// TwinCAT 3 PLC project Plc
// Title: Sample PackML_V2
// Company: Beckhoff Automation GmbH
// Author: Beckhoff Automation GmbH
// ProjectVersion: 3.0.3.0
// Description: Sample PackML_V2
// ProgramVersion: 3.1.0.9
// libraries:
//   CHALET_BaseComponents, * (Beckhoff CH)
//   CHALET_Nc, * (Beckhoff CH)
//   CHALET_Vision, * (Beckhoff CH)
//   CHALET_XPlanar, * (Beckhoff CH)
//   Tc2_ControllerToolbox, * (Beckhoff Automation GmbH)
//   Tc2_EtherCAT, * (Beckhoff Automation GmbH)
//   Tc2_MC2, * (Beckhoff Automation GmbH)
//   Tc2_Standard, * (Beckhoff Automation GmbH)
//   Tc2_System, * (Beckhoff Automation GmbH)
//   Tc2_Utilities, * (Beckhoff Automation GmbH)
//   Tc3_Mc3PlanarMotion, * (Beckhoff Automation GmbH)
//   Tc3_Module, * (Beckhoff Automation GmbH)
//   Tc3_PackML_V2, * (Beckhoff Automation GmbH)
//   Tc3_Vision, * (Beckhoff Automation GmbH)
//   Tc3_XPlanarUtility, * (Beckhoff Automation GmbH & Co. KG)
// project tree:
//   COMPONENTs/ Debug.TcGVL, E_ObservationState.TcDUT, GVL_Components.TcGVL, FB_Machine.TcPOU, FB_RollingAverage_Ppm.TcPOU
//   COMPONENTs/Mode/ E_PMLMode.TcDUT, E_PMLStopReason.TcDUT
//   COMPONENTs/OEE/ ST_Analytics.TcDUT
//   COMPONENTs/PackML/ ST_PMLc_Custom.TcDUT, ST_PMLs_Custom.TcDUT, ST_PML_Custom.TcDUT
//   COMPONENTs/Unit/ FB_Unit.TcPOU
//   COMPONENTs/Vision/ E_VisionState.TcDUT, FB_VsSystem.TcPOU, I_VsSystem_Check.TcIO, I_VsSystem_Plc.TcIO
//   / PlcTask.TcTTO, VisionTask.TcTTO
//   THREADs/ PRG_ProcessCellSimulation.TcPOU, PRG_Vision.TcPOU
// real-time tasks:
//   TASK Task_Plc: cycle T#1ms, priority 5, ADS port 350
//   TASK Task_XPlanar_Hardware: cycle T#250us, priority 1, ADS port 351
//   TASK Task_XPlanar_Execute: cycle T#1ms, priority 3, ADS port 352
//   TASK Task_XPlanar_Prepare: cycle T#10ms, priority 10, ADS port 353
//   TASK Task_Job: cycle default, priority 7
//   TASK Task_Vision_Acquisition: cycle T#1ms, priority 4, ADS port 354
//   TASK Task_Vision_Display: cycle T#10ms, priority 12, ADS port 355
//   TASK Task_Vision_Execute: cycle T#10ms, priority 11, ADS port 356
//   TASK Task_IO: cycle T#50000us, priority 14, ADS port 301
//   TASK PlcTask: cycle T#10ms, priority 20, ADS port 357
//   TASK AnalyticsTask: cycle T#10ms, priority 21, ADS port 358
//   TASK AnalyticsTask_C1: cycle T#10ms, priority 22, ADS port 359
// I/O:
//   DEVICE Device 4 (USB)
//     Box 2 (C9900-L100 License-Key-USB-Stick)
//   DEVICE Device 5 (EtherCAT), AmsNetId 10.16.0.17.6.1
//     Term 1 (EK1100) [EK1100 EtherCAT Coupler (2A E-Bus)]
//       Term 2 (EK1322) [EK1322 2-port EtherCAT P junction with feed-in]
//       Term 3 (EK1322) [EK1322 2-port EtherCAT P junction with feed-in]
//         Box 19 (VCS2001-0500) [VCS2001-0500 | Area scan camera, 2.5 GBit/s, Sony IMX264, color, 5.0 MP]
//           modules: Gerät
//       Term 5 (EK1322) [EK1322 2-port EtherCAT P junction with feed-in]
//         Box 6 (VIP2000-1010) [VIP2000 Flaechenbeleuchtung, OGB-IR850, breitstrahlend, 100 x 100 mm]
//           modules: Device, Channel Infrared, Channel Blue, Channel Green, Channel Orange, Calibration Data, Calibration Data, Calibration Data, Calibration Data, Calibration Data, Calibration Data, Calibration Data, Calibration Data, Calibration Data, Calibration Data, Calibration Data, Calibration Data, Calibration Data, Calibration Data, Calibration Data, Calibration Data, Calibration Data, Calibration Data, Calibration Data, Calibration Data
//         Box 7 (VIP2000-1010) [VIP2000 Flaechenbeleuchtung, OGB-IR850, breitstrahlend, 100 x 100 mm]
//           modules: Device, Channel Infrared, Channel Blue, Channel Green, Channel Orange, Calibration Data, Calibration Data, Calibration Data, Calibration Data, Calibration Data, Calibration Data, Calibration Data, Calibration Data, Calibration Data, Calibration Data, Calibration Data, Calibration Data, Calibration Data, Calibration Data, Calibration Data, Calibration Data, Calibration Data, Calibration Data, Calibration Data, Calibration Data
//       Term 8 (EL9227-5500) [EL9227-5500 Overcurrent protection 24V DC, 2Ch., max. 10A (sum), adjustable, extended functionalities]
//       Term 9 (EL9227-9664) [EL9227-9664 Overcurrent protection 24V DC, 2Ch., 6A/4A, extended functionalities]
//       Term 11 (EL9011) [EL9011 End Terminal]
//     Box 10 (EP2316-0003) [EP2316-0003 8 Ch. Dig. In, 10µs, 8Ch. Dig. Out 24V, 0,5A, Diagnostic, 10-Pole Plug Connector]
//   DEVICE Device 2 (RT-Ethernet Adapter)
//   DEVICE Device 3 (EtherCAT), AmsNetId 10.16.0.17.4.1
//     Term 4 (APS4322-7000) [APS4322-7000 Drive]
//       Term 12 (APS4322-5000) [APS4322-5000 Feedback]
//     Term 13 (APS4322-7000) [APS4322-7000 Drive]
//       Term 14 (APS4322-5000) [APS4322-5000 Feedback]
// variable links:
//   Device 3 (EtherCAT) <-> TcCOM Objects/XPlanar/Part1/Tile1
//     Term 4 (APS4322-7000)/APS Comm Inputs/CommStatusWord <-> Data Pointer/MoverCommStatusWord
//     Term 4 (APS4322-7000)/APS Comm Inputs/Data {1..4} <-> Data Pointer/MoverCommDataIn[{0..3}]  (4 links)
//     Term 4 (APS4322-7000)/APS Comm Outputs/CommControlWord <-> Data Pointer/MoverCommControlWord
//     Term 4 (APS4322-7000)/APS Comm Outputs/Data 1 <-> Data Pointer/MoverCommDataOut
//     Term 4 (APS4322-7000)/APS Diagdata/DC Link Voltage <-> Data Pointer/DcLinkVoltage
//     Term 4 (APS4322-7000)/APS Diagdata/Power supply current <-> Data Pointer/PowerSupplyCurrent
//     Term 4 (APS4322-7000)/APS Inputs/StatusWord <-> Data Pointer/PowerUnitStatusWord
//     Term 4 (APS4322-7000)/APS Outputs/ControlWord <-> Data Pointer/PowerUnitControlWord
//     Term 4 (APS4322-7000)/APS Outputs/Current D 0X0 <-> Data Pointer/DCurrentSetPoints[0]
//     Term 4 (APS4322-7000)/APS Outputs/Current D 0X1 <-> Data Pointer/DCurrentSetPoints[1]
//     Term 4 (APS4322-7000)/APS Outputs/Current D 0X2 <-> Data Pointer/DCurrentSetPoints[2]
//     Term 4 (APS4322-7000)/APS Outputs/Current D 1X0 <-> Data Pointer/DCurrentSetPoints[6]
//     Term 4 (APS4322-7000)/APS Outputs/Current D 1X1 <-> Data Pointer/DCurrentSetPoints[7]
//     Term 4 (APS4322-7000)/APS Outputs/Current D 1X2 <-> Data Pointer/DCurrentSetPoints[8]
//     Term 4 (APS4322-7000)/APS Outputs/Current D 2X0 <-> Data Pointer/DCurrentSetPoints[12]
//     Term 4 (APS4322-7000)/APS Outputs/Current D 2X1 <-> Data Pointer/DCurrentSetPoints[13]
//     Term 4 (APS4322-7000)/APS Outputs/Current D 2X2 <-> Data Pointer/DCurrentSetPoints[14]
//     Term 4 (APS4322-7000)/APS Outputs/Current D 3X0 <-> Data Pointer/DCurrentSetPoints[18]
//     Term 4 (APS4322-7000)/APS Outputs/Current D 3X1 <-> Data Pointer/DCurrentSetPoints[19]
//     Term 4 (APS4322-7000)/APS Outputs/Current D 3X2 <-> Data Pointer/DCurrentSetPoints[20]
//     Term 4 (APS4322-7000)/APS Outputs/Current D 0Y0 <-> Data Pointer/DCurrentSetPoints[3]
//     Term 4 (APS4322-7000)/APS Outputs/Current D 0Y1 <-> Data Pointer/DCurrentSetPoints[4]
//     Term 4 (APS4322-7000)/APS Outputs/Current D 0Y2 <-> Data Pointer/DCurrentSetPoints[5]
//     Term 4 (APS4322-7000)/APS Outputs/Current D 1Y0 <-> Data Pointer/DCurrentSetPoints[9]
//     Term 4 (APS4322-7000)/APS Outputs/Current D 1Y1 <-> Data Pointer/DCurrentSetPoints[10]
//     Term 4 (APS4322-7000)/APS Outputs/Current D 1Y2 <-> Data Pointer/DCurrentSetPoints[11]
//     Term 4 (APS4322-7000)/APS Outputs/Current D 2Y0 <-> Data Pointer/DCurrentSetPoints[15]
//     Term 4 (APS4322-7000)/APS Outputs/Current D 2Y1 <-> Data Pointer/DCurrentSetPoints[16]
//     Term 4 (APS4322-7000)/APS Outputs/Current D 2Y2 <-> Data Pointer/DCurrentSetPoints[17]
//     Term 4 (APS4322-7000)/APS Outputs/Current D 3Y0 <-> Data Pointer/DCurrentSetPoints[21]
//     Term 4 (APS4322-7000)/APS Outputs/Current D 3Y1 <-> Data Pointer/DCurrentSetPoints[22]
//     Term 4 (APS4322-7000)/APS Outputs/Current D 3Y2 <-> Data Pointer/DCurrentSetPoints[23]
//     Term 4 (APS4322-7000)/APS Outputs/Current Q 0X0 <-> Data Pointer/QCurrentSetPoints[0]
//     Term 4 (APS4322-7000)/APS Outputs/Current Q 0X1 <-> Data Pointer/QCurrentSetPoints[1]
//     Term 4 (APS4322-7000)/APS Outputs/Current Q 0X2 <-> Data Pointer/QCurrentSetPoints[2]
//     Term 4 (APS4322-7000)/APS Outputs/Current Q 1X0 <-> Data Pointer/QCurrentSetPoints[6]
//     Term 4 (APS4322-7000)/APS Outputs/Current Q 1X1 <-> Data Pointer/QCurrentSetPoints[7]
//     Term 4 (APS4322-7000)/APS Outputs/Current Q 1X2 <-> Data Pointer/QCurrentSetPoints[8]
//     Term 4 (APS4322-7000)/APS Outputs/Current Q 2X0 <-> Data Pointer/QCurrentSetPoints[12]
//     Term 4 (APS4322-7000)/APS Outputs/Current Q 2X1 <-> Data Pointer/QCurrentSetPoints[13]
//     Term 4 (APS4322-7000)/APS Outputs/Current Q 2X2 <-> Data Pointer/QCurrentSetPoints[14]
//     Term 4 (APS4322-7000)/APS Outputs/Current Q 3X0 <-> Data Pointer/QCurrentSetPoints[18]
//     Term 4 (APS4322-7000)/APS Outputs/Current Q 3X1 <-> Data Pointer/QCurrentSetPoints[19]
//     Term 4 (APS4322-7000)/APS Outputs/Current Q 3X2 <-> Data Pointer/QCurrentSetPoints[20]
//     Term 4 (APS4322-7000)/APS Outputs/Current Q 0Y0 <-> Data Pointer/QCurrentSetPoints[3]
//     Term 4 (APS4322-7000)/APS Outputs/Current Q 0Y1 <-> Data Pointer/QCurrentSetPoints[4]
//     Term 4 (APS4322-7000)/APS Outputs/Current Q 0Y2 <-> Data Pointer/QCurrentSetPoints[5]
//     Term 4 (APS4322-7000)/APS Outputs/Current Q 1Y0 <-> Data Pointer/QCurrentSetPoints[9]
//     Term 4 (APS4322-7000)/APS Outputs/Current Q 1Y1 <-> Data Pointer/QCurrentSetPoints[10]
//     Term 4 (APS4322-7000)/APS Outputs/Current Q 1Y2 <-> Data Pointer/QCurrentSetPoints[11]
//     Term 4 (APS4322-7000)/APS Outputs/Current Q 2Y0 <-> Data Pointer/QCurrentSetPoints[15]
//     Term 4 (APS4322-7000)/APS Outputs/Current Q 2Y1 <-> Data Pointer/QCurrentSetPoints[16]
//     Term 4 (APS4322-7000)/APS Outputs/Current Q 2Y2 <-> Data Pointer/QCurrentSetPoints[17]
//     Term 4 (APS4322-7000)/APS Outputs/Current Q 3Y0 <-> Data Pointer/QCurrentSetPoints[21]
//     Term 4 (APS4322-7000)/APS Outputs/Current Q 3Y1 <-> Data Pointer/QCurrentSetPoints[22]
//     Term 4 (APS4322-7000)/APS Outputs/Current Q 3Y2 <-> Data Pointer/QCurrentSetPoints[23]
//     Term 4 (APS4322-7000)/APS Outputs/PhiE 0X0 <-> Data Pointer/PhiSetPoints[0]
//     Term 4 (APS4322-7000)/APS Outputs/PhiE 0X1 <-> Data Pointer/PhiSetPoints[1]
//     Term 4 (APS4322-7000)/APS Outputs/PhiE 0X2 <-> Data Pointer/PhiSetPoints[2]
//     Term 4 (APS4322-7000)/APS Outputs/PhiE 1X0 <-> Data Pointer/PhiSetPoints[6]
//     Term 4 (APS4322-7000)/APS Outputs/PhiE 1X1 <-> Data Pointer/PhiSetPoints[7]
//     Term 4 (APS4322-7000)/APS Outputs/PhiE 1X2 <-> Data Pointer/PhiSetPoints[8]
//     Term 4 (APS4322-7000)/APS Outputs/PhiE 2X0 <-> Data Pointer/PhiSetPoints[12]
//     Term 4 (APS4322-7000)/APS Outputs/PhiE 2X1 <-> Data Pointer/PhiSetPoints[13]
//     Term 4 (APS4322-7000)/APS Outputs/PhiE 2X2 <-> Data Pointer/PhiSetPoints[14]
//     Term 4 (APS4322-7000)/APS Outputs/PhiE 3X0 <-> Data Pointer/PhiSetPoints[18]
//     Term 4 (APS4322-7000)/APS Outputs/PhiE 3X1 <-> Data Pointer/PhiSetPoints[19]
//     Term 4 (APS4322-7000)/APS Outputs/PhiE 3X2 <-> Data Pointer/PhiSetPoints[20]
//     Term 4 (APS4322-7000)/APS Outputs/PhiE 0Y0 <-> Data Pointer/PhiSetPoints[3]
//     Term 4 (APS4322-7000)/APS Outputs/PhiE 0Y1 <-> Data Pointer/PhiSetPoints[4]
//     Term 4 (APS4322-7000)/APS Outputs/PhiE 0Y2 <-> Data Pointer/PhiSetPoints[5]
//     Term 4 (APS4322-7000)/APS Outputs/PhiE 1Y0 <-> Data Pointer/PhiSetPoints[9]
//     Term 4 (APS4322-7000)/APS Outputs/PhiE 1Y1 <-> Data Pointer/PhiSetPoints[10]
//     Term 4 (APS4322-7000)/APS Outputs/PhiE 1Y2 <-> Data Pointer/PhiSetPoints[11]
//     Term 4 (APS4322-7000)/APS Outputs/PhiE 2Y0 <-> Data Pointer/PhiSetPoints[15]
//     Term 4 (APS4322-7000)/APS Outputs/PhiE 2Y1 <-> Data Pointer/PhiSetPoints[16]
//     Term 4 (APS4322-7000)/APS Outputs/PhiE 2Y2 <-> Data Pointer/PhiSetPoints[17]
//     Term 4 (APS4322-7000)/APS Outputs/PhiE 3Y0 <-> Data Pointer/PhiSetPoints[21]
//     Term 4 (APS4322-7000)/APS Outputs/PhiE 3Y1 <-> Data Pointer/PhiSetPoints[22]
//     Term 4 (APS4322-7000)/APS Outputs/PhiE 3Y2 <-> Data Pointer/PhiSetPoints[23]
//     Term 4 (APS4322-7000)/Term 12 (APS4322-5000)/FB Inputs/A{0..8 step 2} X-Field <-> Data Pointer/HallSensorFieldsXYZ[{0..12 step 3}]  (5 links)
//     Term 4 (APS4322-7000)/Term 12 (APS4322-5000)/FB Inputs/A{0..8 step 2} Y-Field <-> Data Pointer/HallSensorFieldsXYZ[{1..13 step 3}]  (5 links)
//     Term 4 (APS4322-7000)/Term 12 (APS4322-5000)/FB Inputs/A{0..8 step 2} Z-Field <-> Data Pointer/HallSensorFieldsXYZ[{2..14 step 3}]  (5 links)
//     Term 4 (APS4322-7000)/Term 12 (APS4322-5000)/FB Inputs/B{1..9 step 2} X-Field <-> Data Pointer/HallSensorFieldsXYZ[{15..27 step 3}]  (5 links)
//     Term 4 (APS4322-7000)/Term 12 (APS4322-5000)/FB Inputs/B{1..9 step 2} Y-Field <-> Data Pointer/HallSensorFieldsXYZ[{16..28 step 3}]  (5 links)
//     Term 4 (APS4322-7000)/Term 12 (APS4322-5000)/FB Inputs/B{1..9 step 2} Z-Field <-> Data Pointer/HallSensorFieldsXYZ[{17..29 step 3}]  (5 links)
//     Term 4 (APS4322-7000)/Term 12 (APS4322-5000)/FB Inputs/C{0..8 step 2} X-Field <-> Data Pointer/HallSensorFieldsXYZ[{30..42 step 3}]  (5 links)
//     Term 4 (APS4322-7000)/Term 12 (APS4322-5000)/FB Inputs/C{0..8 step 2} Y-Field <-> Data Pointer/HallSensorFieldsXYZ[{31..43 step 3}]  (5 links)
//     Term 4 (APS4322-7000)/Term 12 (APS4322-5000)/FB Inputs/C{0..8 step 2} Z-Field <-> Data Pointer/HallSensorFieldsXYZ[{32..44 step 3}]  (5 links)
//     Term 4 (APS4322-7000)/Term 12 (APS4322-5000)/FB Inputs/D{1..9 step 2} X-Field <-> Data Pointer/HallSensorFieldsXYZ[{45..57 step 3}]  (5 links)
//     Term 4 (APS4322-7000)/Term 12 (APS4322-5000)/FB Inputs/D{1..9 step 2} Y-Field <-> Data Pointer/HallSensorFieldsXYZ[{46..58 step 3}]  (5 links)
//     Term 4 (APS4322-7000)/Term 12 (APS4322-5000)/FB Inputs/D{1..9 step 2} Z-Field <-> Data Pointer/HallSensorFieldsXYZ[{47..59 step 3}]  (5 links)
//     Term 4 (APS4322-7000)/Term 12 (APS4322-5000)/FB Inputs/E{0..8 step 2} X-Field <-> Data Pointer/HallSensorFieldsXYZ[{60..72 step 3}]  (5 links)
//     Term 4 (APS4322-7000)/Term 12 (APS4322-5000)/FB Inputs/E{0..8 step 2} Y-Field <-> Data Pointer/HallSensorFieldsXYZ[{61..73 step 3}]  (5 links)
//     Term 4 (APS4322-7000)/Term 12 (APS4322-5000)/FB Inputs/E{0..8 step 2} Z-Field <-> Data Pointer/HallSensorFieldsXYZ[{62..74 step 3}]  (5 links)
//     Term 4 (APS4322-7000)/Term 12 (APS4322-5000)/FB Inputs/F{1..9 step 2} X-Field <-> Data Pointer/HallSensorFieldsXYZ[{75..87 step 3}]  (5 links)
//     Term 4 (APS4322-7000)/Term 12 (APS4322-5000)/FB Inputs/F{1..9 step 2} Y-Field <-> Data Pointer/HallSensorFieldsXYZ[{76..88 step 3}]  (5 links)
//     Term 4 (APS4322-7000)/Term 12 (APS4322-5000)/FB Inputs/F{1..9 step 2} Z-Field <-> Data Pointer/HallSensorFieldsXYZ[{77..89 step 3}]  (5 links)
//     Term 4 (APS4322-7000)/Term 12 (APS4322-5000)/FB Inputs/G{0..8 step 2} X-Field <-> Data Pointer/HallSensorFieldsXYZ[{90..102 step 3}]  (5 links)
//     Term 4 (APS4322-7000)/Term 12 (APS4322-5000)/FB Inputs/G{0..8 step 2} Y-Field <-> Data Pointer/HallSensorFieldsXYZ[{91..103 step 3}]  (5 links)
//     Term 4 (APS4322-7000)/Term 12 (APS4322-5000)/FB Inputs/G{0..8 step 2} Z-Field <-> Data Pointer/HallSensorFieldsXYZ[{92..104 step 3}]  (5 links)
//     Term 4 (APS4322-7000)/Term 12 (APS4322-5000)/FB Inputs/H{1..9 step 2} X-Field <-> Data Pointer/HallSensorFieldsXYZ[{105..117 step 3}]  (5 links)
//     Term 4 (APS4322-7000)/Term 12 (APS4322-5000)/FB Inputs/H{1..9 step 2} Y-Field <-> Data Pointer/HallSensorFieldsXYZ[{106..118 step 3}]  (5 links)
//     Term 4 (APS4322-7000)/Term 12 (APS4322-5000)/FB Inputs/H{1..9 step 2} Z-Field <-> Data Pointer/HallSensorFieldsXYZ[{107..119 step 3}]  (5 links)
//     Term 4 (APS4322-7000)/Term 12 (APS4322-5000)/FB Inputs/I{0..8 step 2} X-Field <-> Data Pointer/HallSensorFieldsXYZ[{120..132 step 3}]  (5 links)
//     Term 4 (APS4322-7000)/Term 12 (APS4322-5000)/FB Inputs/I{0..8 step 2} Y-Field <-> Data Pointer/HallSensorFieldsXYZ[{121..133 step 3}]  (5 links)
//     Term 4 (APS4322-7000)/Term 12 (APS4322-5000)/FB Inputs/I{0..8 step 2} Z-Field <-> Data Pointer/HallSensorFieldsXYZ[{122..134 step 3}]  (5 links)
//     Term 4 (APS4322-7000)/Term 12 (APS4322-5000)/FB Inputs/J{1..9 step 2} X-Field <-> Data Pointer/HallSensorFieldsXYZ[{135..147 step 3}]  (5 links)
//     Term 4 (APS4322-7000)/Term 12 (APS4322-5000)/FB Inputs/J{1..9 step 2} Y-Field <-> Data Pointer/HallSensorFieldsXYZ[{136..148 step 3}]  (5 links)
//     Term 4 (APS4322-7000)/Term 12 (APS4322-5000)/FB Inputs/J{1..9 step 2} Z-Field <-> Data Pointer/HallSensorFieldsXYZ[{137..149 step 3}]  (5 links)
//     Term 4 (APS4322-7000)/Term 12 (APS4322-5000)/FB Inputs/Status <-> Data Pointer/FeedbackStatus
//   Device 3 (EtherCAT) <-> TcCOM Objects/XPlanar/Part1/Tile2
//     Term 13 (APS4322-7000)/APS Comm Inputs/CommStatusWord <-> Data Pointer/MoverCommStatusWord
//     Term 13 (APS4322-7000)/APS Comm Inputs/Data {1..4} <-> Data Pointer/MoverCommDataIn[{0..3}]  (4 links)
//     Term 13 (APS4322-7000)/APS Comm Outputs/CommControlWord <-> Data Pointer/MoverCommControlWord
//     Term 13 (APS4322-7000)/APS Comm Outputs/Data 1 <-> Data Pointer/MoverCommDataOut
//     Term 13 (APS4322-7000)/APS Diagdata/DC Link Voltage <-> Data Pointer/DcLinkVoltage
//     Term 13 (APS4322-7000)/APS Diagdata/Power supply current <-> Data Pointer/PowerSupplyCurrent
//     Term 13 (APS4322-7000)/APS Inputs/StatusWord <-> Data Pointer/PowerUnitStatusWord
//     Term 13 (APS4322-7000)/APS Outputs/ControlWord <-> Data Pointer/PowerUnitControlWord
//     Term 13 (APS4322-7000)/APS Outputs/Current D 0X0 <-> Data Pointer/DCurrentSetPoints[0]
//     Term 13 (APS4322-7000)/APS Outputs/Current D 0X1 <-> Data Pointer/DCurrentSetPoints[1]
//     Term 13 (APS4322-7000)/APS Outputs/Current D 0X2 <-> Data Pointer/DCurrentSetPoints[2]
//     Term 13 (APS4322-7000)/APS Outputs/Current D 1X0 <-> Data Pointer/DCurrentSetPoints[6]
//     Term 13 (APS4322-7000)/APS Outputs/Current D 1X1 <-> Data Pointer/DCurrentSetPoints[7]
//     Term 13 (APS4322-7000)/APS Outputs/Current D 1X2 <-> Data Pointer/DCurrentSetPoints[8]
//     Term 13 (APS4322-7000)/APS Outputs/Current D 2X0 <-> Data Pointer/DCurrentSetPoints[12]
//     Term 13 (APS4322-7000)/APS Outputs/Current D 2X1 <-> Data Pointer/DCurrentSetPoints[13]
//     Term 13 (APS4322-7000)/APS Outputs/Current D 2X2 <-> Data Pointer/DCurrentSetPoints[14]
//     Term 13 (APS4322-7000)/APS Outputs/Current D 3X0 <-> Data Pointer/DCurrentSetPoints[18]
//     Term 13 (APS4322-7000)/APS Outputs/Current D 3X1 <-> Data Pointer/DCurrentSetPoints[19]
//     Term 13 (APS4322-7000)/APS Outputs/Current D 3X2 <-> Data Pointer/DCurrentSetPoints[20]
//     Term 13 (APS4322-7000)/APS Outputs/Current D 0Y0 <-> Data Pointer/DCurrentSetPoints[3]
//     Term 13 (APS4322-7000)/APS Outputs/Current D 0Y1 <-> Data Pointer/DCurrentSetPoints[4]
//     Term 13 (APS4322-7000)/APS Outputs/Current D 0Y2 <-> Data Pointer/DCurrentSetPoints[5]
//     Term 13 (APS4322-7000)/APS Outputs/Current D 1Y0 <-> Data Pointer/DCurrentSetPoints[9]
//     Term 13 (APS4322-7000)/APS Outputs/Current D 1Y1 <-> Data Pointer/DCurrentSetPoints[10]
//     Term 13 (APS4322-7000)/APS Outputs/Current D 1Y2 <-> Data Pointer/DCurrentSetPoints[11]
//     Term 13 (APS4322-7000)/APS Outputs/Current D 2Y0 <-> Data Pointer/DCurrentSetPoints[15]
//     Term 13 (APS4322-7000)/APS Outputs/Current D 2Y1 <-> Data Pointer/DCurrentSetPoints[16]
//     Term 13 (APS4322-7000)/APS Outputs/Current D 2Y2 <-> Data Pointer/DCurrentSetPoints[17]
//     Term 13 (APS4322-7000)/APS Outputs/Current D 3Y0 <-> Data Pointer/DCurrentSetPoints[21]
//     Term 13 (APS4322-7000)/APS Outputs/Current D 3Y1 <-> Data Pointer/DCurrentSetPoints[22]
//     Term 13 (APS4322-7000)/APS Outputs/Current D 3Y2 <-> Data Pointer/DCurrentSetPoints[23]
//     Term 13 (APS4322-7000)/APS Outputs/Current Q 0X0 <-> Data Pointer/QCurrentSetPoints[0]
//     Term 13 (APS4322-7000)/APS Outputs/Current Q 0X1 <-> Data Pointer/QCurrentSetPoints[1]
//     Term 13 (APS4322-7000)/APS Outputs/Current Q 0X2 <-> Data Pointer/QCurrentSetPoints[2]
//     Term 13 (APS4322-7000)/APS Outputs/Current Q 1X0 <-> Data Pointer/QCurrentSetPoints[6]
//     Term 13 (APS4322-7000)/APS Outputs/Current Q 1X1 <-> Data Pointer/QCurrentSetPoints[7]
//     Term 13 (APS4322-7000)/APS Outputs/Current Q 1X2 <-> Data Pointer/QCurrentSetPoints[8]
//     Term 13 (APS4322-7000)/APS Outputs/Current Q 2X0 <-> Data Pointer/QCurrentSetPoints[12]
//     Term 13 (APS4322-7000)/APS Outputs/Current Q 2X1 <-> Data Pointer/QCurrentSetPoints[13]
//     Term 13 (APS4322-7000)/APS Outputs/Current Q 2X2 <-> Data Pointer/QCurrentSetPoints[14]
//     Term 13 (APS4322-7000)/APS Outputs/Current Q 3X0 <-> Data Pointer/QCurrentSetPoints[18]
//     Term 13 (APS4322-7000)/APS Outputs/Current Q 3X1 <-> Data Pointer/QCurrentSetPoints[19]
//     Term 13 (APS4322-7000)/APS Outputs/Current Q 3X2 <-> Data Pointer/QCurrentSetPoints[20]
//     Term 13 (APS4322-7000)/APS Outputs/Current Q 0Y0 <-> Data Pointer/QCurrentSetPoints[3]
//     Term 13 (APS4322-7000)/APS Outputs/Current Q 0Y1 <-> Data Pointer/QCurrentSetPoints[4]
//     Term 13 (APS4322-7000)/APS Outputs/Current Q 0Y2 <-> Data Pointer/QCurrentSetPoints[5]
//     Term 13 (APS4322-7000)/APS Outputs/Current Q 1Y0 <-> Data Pointer/QCurrentSetPoints[9]
//     Term 13 (APS4322-7000)/APS Outputs/Current Q 1Y1 <-> Data Pointer/QCurrentSetPoints[10]
//     Term 13 (APS4322-7000)/APS Outputs/Current Q 1Y2 <-> Data Pointer/QCurrentSetPoints[11]
//     Term 13 (APS4322-7000)/APS Outputs/Current Q 2Y0 <-> Data Pointer/QCurrentSetPoints[15]
//     Term 13 (APS4322-7000)/APS Outputs/Current Q 2Y1 <-> Data Pointer/QCurrentSetPoints[16]
//     Term 13 (APS4322-7000)/APS Outputs/Current Q 2Y2 <-> Data Pointer/QCurrentSetPoints[17]
//     Term 13 (APS4322-7000)/APS Outputs/Current Q 3Y0 <-> Data Pointer/QCurrentSetPoints[21]
//     Term 13 (APS4322-7000)/APS Outputs/Current Q 3Y1 <-> Data Pointer/QCurrentSetPoints[22]
//     Term 13 (APS4322-7000)/APS Outputs/Current Q 3Y2 <-> Data Pointer/QCurrentSetPoints[23]
//     Term 13 (APS4322-7000)/APS Outputs/PhiE 0X0 <-> Data Pointer/PhiSetPoints[0]
//     Term 13 (APS4322-7000)/APS Outputs/PhiE 0X1 <-> Data Pointer/PhiSetPoints[1]
//     Term 13 (APS4322-7000)/APS Outputs/PhiE 0X2 <-> Data Pointer/PhiSetPoints[2]
//     Term 13 (APS4322-7000)/APS Outputs/PhiE 1X0 <-> Data Pointer/PhiSetPoints[6]
//     Term 13 (APS4322-7000)/APS Outputs/PhiE 1X1 <-> Data Pointer/PhiSetPoints[7]
//     Term 13 (APS4322-7000)/APS Outputs/PhiE 1X2 <-> Data Pointer/PhiSetPoints[8]
//     Term 13 (APS4322-7000)/APS Outputs/PhiE 2X0 <-> Data Pointer/PhiSetPoints[12]
//     Term 13 (APS4322-7000)/APS Outputs/PhiE 2X1 <-> Data Pointer/PhiSetPoints[13]
//     Term 13 (APS4322-7000)/APS Outputs/PhiE 2X2 <-> Data Pointer/PhiSetPoints[14]
//     Term 13 (APS4322-7000)/APS Outputs/PhiE 3X0 <-> Data Pointer/PhiSetPoints[18]
//     Term 13 (APS4322-7000)/APS Outputs/PhiE 3X1 <-> Data Pointer/PhiSetPoints[19]
//     Term 13 (APS4322-7000)/APS Outputs/PhiE 3X2 <-> Data Pointer/PhiSetPoints[20]
//     Term 13 (APS4322-7000)/APS Outputs/PhiE 0Y0 <-> Data Pointer/PhiSetPoints[3]
//     Term 13 (APS4322-7000)/APS Outputs/PhiE 0Y1 <-> Data Pointer/PhiSetPoints[4]
//     Term 13 (APS4322-7000)/APS Outputs/PhiE 0Y2 <-> Data Pointer/PhiSetPoints[5]
//     Term 13 (APS4322-7000)/APS Outputs/PhiE 1Y0 <-> Data Pointer/PhiSetPoints[9]
//     Term 13 (APS4322-7000)/APS Outputs/PhiE 1Y1 <-> Data Pointer/PhiSetPoints[10]
//     Term 13 (APS4322-7000)/APS Outputs/PhiE 1Y2 <-> Data Pointer/PhiSetPoints[11]
//     Term 13 (APS4322-7000)/APS Outputs/PhiE 2Y0 <-> Data Pointer/PhiSetPoints[15]
//     Term 13 (APS4322-7000)/APS Outputs/PhiE 2Y1 <-> Data Pointer/PhiSetPoints[16]
//     Term 13 (APS4322-7000)/APS Outputs/PhiE 2Y2 <-> Data Pointer/PhiSetPoints[17]
//     Term 13 (APS4322-7000)/APS Outputs/PhiE 3Y0 <-> Data Pointer/PhiSetPoints[21]
//     Term 13 (APS4322-7000)/APS Outputs/PhiE 3Y1 <-> Data Pointer/PhiSetPoints[22]
//     Term 13 (APS4322-7000)/APS Outputs/PhiE 3Y2 <-> Data Pointer/PhiSetPoints[23]
//     Term 13 (APS4322-7000)/Term 14 (APS4322-5000)/FB Inputs/A{0..8 step 2} X-Field <-> Data Pointer/HallSensorFieldsXYZ[{0..12 step 3}]  (5 links)
//     Term 13 (APS4322-7000)/Term 14 (APS4322-5000)/FB Inputs/A{0..8 step 2} Y-Field <-> Data Pointer/HallSensorFieldsXYZ[{1..13 step 3}]  (5 links)
//     Term 13 (APS4322-7000)/Term 14 (APS4322-5000)/FB Inputs/A{0..8 step 2} Z-Field <-> Data Pointer/HallSensorFieldsXYZ[{2..14 step 3}]  (5 links)
//     Term 13 (APS4322-7000)/Term 14 (APS4322-5000)/FB Inputs/B{1..9 step 2} X-Field <-> Data Pointer/HallSensorFieldsXYZ[{15..27 step 3}]  (5 links)
//     Term 13 (APS4322-7000)/Term 14 (APS4322-5000)/FB Inputs/B{1..9 step 2} Y-Field <-> Data Pointer/HallSensorFieldsXYZ[{16..28 step 3}]  (5 links)
//     Term 13 (APS4322-7000)/Term 14 (APS4322-5000)/FB Inputs/B{1..9 step 2} Z-Field <-> Data Pointer/HallSensorFieldsXYZ[{17..29 step 3}]  (5 links)
//     Term 13 (APS4322-7000)/Term 14 (APS4322-5000)/FB Inputs/C{0..8 step 2} X-Field <-> Data Pointer/HallSensorFieldsXYZ[{30..42 step 3}]  (5 links)
//     Term 13 (APS4322-7000)/Term 14 (APS4322-5000)/FB Inputs/C{0..8 step 2} Y-Field <-> Data Pointer/HallSensorFieldsXYZ[{31..43 step 3}]  (5 links)
//     Term 13 (APS4322-7000)/Term 14 (APS4322-5000)/FB Inputs/C{0..8 step 2} Z-Field <-> Data Pointer/HallSensorFieldsXYZ[{32..44 step 3}]  (5 links)
//     Term 13 (APS4322-7000)/Term 14 (APS4322-5000)/FB Inputs/D{1..9 step 2} X-Field <-> Data Pointer/HallSensorFieldsXYZ[{45..57 step 3}]  (5 links)
//     Term 13 (APS4322-7000)/Term 14 (APS4322-5000)/FB Inputs/D{1..9 step 2} Y-Field <-> Data Pointer/HallSensorFieldsXYZ[{46..58 step 3}]  (5 links)
//     Term 13 (APS4322-7000)/Term 14 (APS4322-5000)/FB Inputs/D{1..9 step 2} Z-Field <-> Data Pointer/HallSensorFieldsXYZ[{47..59 step 3}]  (5 links)
//     Term 13 (APS4322-7000)/Term 14 (APS4322-5000)/FB Inputs/E{0..8 step 2} X-Field <-> Data Pointer/HallSensorFieldsXYZ[{60..72 step 3}]  (5 links)
//     Term 13 (APS4322-7000)/Term 14 (APS4322-5000)/FB Inputs/E{0..8 step 2} Y-Field <-> Data Pointer/HallSensorFieldsXYZ[{61..73 step 3}]  (5 links)
//     Term 13 (APS4322-7000)/Term 14 (APS4322-5000)/FB Inputs/E{0..8 step 2} Z-Field <-> Data Pointer/HallSensorFieldsXYZ[{62..74 step 3}]  (5 links)
//     Term 13 (APS4322-7000)/Term 14 (APS4322-5000)/FB Inputs/F{1..9 step 2} X-Field <-> Data Pointer/HallSensorFieldsXYZ[{75..87 step 3}]  (5 links)
//     Term 13 (APS4322-7000)/Term 14 (APS4322-5000)/FB Inputs/F{1..9 step 2} Y-Field <-> Data Pointer/HallSensorFieldsXYZ[{76..88 step 3}]  (5 links)
//     Term 13 (APS4322-7000)/Term 14 (APS4322-5000)/FB Inputs/F{1..9 step 2} Z-Field <-> Data Pointer/HallSensorFieldsXYZ[{77..89 step 3}]  (5 links)
//     Term 13 (APS4322-7000)/Term 14 (APS4322-5000)/FB Inputs/G{0..8 step 2} X-Field <-> Data Pointer/HallSensorFieldsXYZ[{90..102 step 3}]  (5 links)
//     Term 13 (APS4322-7000)/Term 14 (APS4322-5000)/FB Inputs/G{0..8 step 2} Y-Field <-> Data Pointer/HallSensorFieldsXYZ[{91..103 step 3}]  (5 links)
//     Term 13 (APS4322-7000)/Term 14 (APS4322-5000)/FB Inputs/G{0..8 step 2} Z-Field <-> Data Pointer/HallSensorFieldsXYZ[{92..104 step 3}]  (5 links)
//     Term 13 (APS4322-7000)/Term 14 (APS4322-5000)/FB Inputs/H{1..9 step 2} X-Field <-> Data Pointer/HallSensorFieldsXYZ[{105..117 step 3}]  (5 links)
//     Term 13 (APS4322-7000)/Term 14 (APS4322-5000)/FB Inputs/H{1..9 step 2} Y-Field <-> Data Pointer/HallSensorFieldsXYZ[{106..118 step 3}]  (5 links)
//     Term 13 (APS4322-7000)/Term 14 (APS4322-5000)/FB Inputs/H{1..9 step 2} Z-Field <-> Data Pointer/HallSensorFieldsXYZ[{107..119 step 3}]  (5 links)
//     Term 13 (APS4322-7000)/Term 14 (APS4322-5000)/FB Inputs/I{0..8 step 2} X-Field <-> Data Pointer/HallSensorFieldsXYZ[{120..132 step 3}]  (5 links)
//     Term 13 (APS4322-7000)/Term 14 (APS4322-5000)/FB Inputs/I{0..8 step 2} Y-Field <-> Data Pointer/HallSensorFieldsXYZ[{121..133 step 3}]  (5 links)
//     Term 13 (APS4322-7000)/Term 14 (APS4322-5000)/FB Inputs/I{0..8 step 2} Z-Field <-> Data Pointer/HallSensorFieldsXYZ[{122..134 step 3}]  (5 links)
//     Term 13 (APS4322-7000)/Term 14 (APS4322-5000)/FB Inputs/J{1..9 step 2} X-Field <-> Data Pointer/HallSensorFieldsXYZ[{135..147 step 3}]  (5 links)
//     Term 13 (APS4322-7000)/Term 14 (APS4322-5000)/FB Inputs/J{1..9 step 2} Y-Field <-> Data Pointer/HallSensorFieldsXYZ[{136..148 step 3}]  (5 links)
//     Term 13 (APS4322-7000)/Term 14 (APS4322-5000)/FB Inputs/J{1..9 step 2} Z-Field <-> Data Pointer/HallSensorFieldsXYZ[{137..149 step 3}]  (5 links)
//     Term 13 (APS4322-7000)/Term 14 (APS4322-5000)/FB Inputs/Status <-> Data Pointer/FeedbackStatus
//   XPlanar MC Project/Axes/Mover4220_1 <-> TcCOM Objects/XPlanar/Mover4220_1
//     IoToMc/STD <-> OutputsToNC3/HWToNC3
//   Plc/Plc Instance <-> Device 5 (EtherCAT)/Term 1 (EK1100)/Term 3 (EK1322)/Box 19 (VCS2001-0500)
//     PlcTask Outputs/GVL_Components.fbMachine.fbVsSystem.fbCameraTriggerController.nStartTime <-> Gerät/DC Timestamp/GVL_Components.fbMachine.fbVsSystem.fbCameraTriggerController.nStartTime
//   Plc/Plc Instance <-> Device 5 (EtherCAT)/Term 1 (EK1100)/Term 5 (EK1322)/Box 6 (VIP2000-1010)
//     PlcTask Inputs/GVL_Components.fbMachine.fbVsSystem.fbIllumination1.DeviceInputs/bDiag <-> VIMN Inputs Device/bDiag
//     PlcTask Inputs/GVL_Components.fbMachine.fbVsSystem.fbIllumination1.DeviceInputs/bError <-> VIMN Inputs Device/bError
//     PlcTask Inputs/GVL_Components.fbMachine.fbVsSystem.fbIllumination1.DeviceInputs/bReady <-> VIMN Inputs Device/bReady
//     PlcTask Inputs/GVL_Components.fbMachine.fbVsSystem.fbIllumination1.DeviceInputs/bWarning <-> VIMN Inputs Device/bWarning
//     PlcTask Inputs/GVL_Components.fbMachine.fbVsSystem.fbIllumination1.DeviceInputs/nSwitch_on_counter <-> VIMN Inputs Device/nSwitch_on_counter
//     PlcTask Outputs/GVL_Components.fbMachine.fbVsSystem.fbIllumination1.ChannelBlue/nBrightness <-> Channel Blue/VICH_PULSE Outputs/nBrightness
//     PlcTask Outputs/GVL_Components.fbMachine.fbVsSystem.fbIllumination1.ChannelBlue/nDuration_1us <-> Channel Blue/VICH_PULSE Outputs/nDuration_1us
//     PlcTask Outputs/GVL_Components.fbMachine.fbVsSystem.fbIllumination1.ChannelGreen/nBrightness <-> Channel Green/VICH_PULSE Outputs/nBrightness
//     PlcTask Outputs/GVL_Components.fbMachine.fbVsSystem.fbIllumination1.ChannelGreen/nDuration_1us <-> Channel Green/VICH_PULSE Outputs/nDuration_1us
//     PlcTask Outputs/GVL_Components.fbMachine.fbVsSystem.fbIllumination1.ChannelInfrared/nBrightness <-> Channel Infrared/VICH_PULSE Outputs/nBrightness
//     PlcTask Outputs/GVL_Components.fbMachine.fbVsSystem.fbIllumination1.ChannelInfrared/nDuration_1us <-> Channel Infrared/VICH_PULSE Outputs/nDuration_1us
//     PlcTask Outputs/GVL_Components.fbMachine.fbVsSystem.fbIllumination1.ChannelOrange/nBrightness <-> Channel Orange/VICH_PULSE Outputs/nBrightness
//     PlcTask Outputs/GVL_Components.fbMachine.fbVsSystem.fbIllumination1.ChannelOrange/nDuration_1us <-> Channel Orange/VICH_PULSE Outputs/nDuration_1us
//     PlcTask Outputs/GVL_Components.fbMachine.fbVsSystem.fbIllumination1.DeviceOutputs/bEnable <-> VIMN Outputs Device/bEnable
//     PlcTask Outputs/GVL_Components.fbMachine.fbVsSystem.fbIllumination1.DeviceOutputs/bReset <-> VIMN Outputs Device/bReset
//     PlcTask Outputs/GVL_Components.fbMachine.fbVsSystem.fbIllumination1.Pulse_DC_Outputs/nTimestamp <-> Device/VIOM_PULSE_DC Outputs/nTimestamp
//   Plc/Plc Instance <-> Device 5 (EtherCAT)/Term 1 (EK1100)/Term 5 (EK1322)/Box 7 (VIP2000-1010)
//     PlcTask Inputs/GVL_Components.fbMachine.fbVsSystem.fbIllumination2.DeviceInputs/bDiag <-> VIMN Inputs Device/bDiag
//     PlcTask Inputs/GVL_Components.fbMachine.fbVsSystem.fbIllumination2.DeviceInputs/bError <-> VIMN Inputs Device/bError
//     PlcTask Inputs/GVL_Components.fbMachine.fbVsSystem.fbIllumination2.DeviceInputs/bReady <-> VIMN Inputs Device/bReady
//     PlcTask Inputs/GVL_Components.fbMachine.fbVsSystem.fbIllumination2.DeviceInputs/bWarning <-> VIMN Inputs Device/bWarning
//     PlcTask Inputs/GVL_Components.fbMachine.fbVsSystem.fbIllumination2.DeviceInputs/nSwitch_on_counter <-> VIMN Inputs Device/nSwitch_on_counter
//     PlcTask Outputs/GVL_Components.fbMachine.fbVsSystem.fbIllumination2.ChannelBlue/nBrightness <-> Channel Blue/VICH_PULSE Outputs/nBrightness
//     PlcTask Outputs/GVL_Components.fbMachine.fbVsSystem.fbIllumination2.ChannelBlue/nDuration_1us <-> Channel Blue/VICH_PULSE Outputs/nDuration_1us
//     PlcTask Outputs/GVL_Components.fbMachine.fbVsSystem.fbIllumination2.ChannelGreen/nBrightness <-> Channel Green/VICH_PULSE Outputs/nBrightness
//     PlcTask Outputs/GVL_Components.fbMachine.fbVsSystem.fbIllumination2.ChannelGreen/nDuration_1us <-> Channel Green/VICH_PULSE Outputs/nDuration_1us
//     PlcTask Outputs/GVL_Components.fbMachine.fbVsSystem.fbIllumination2.ChannelInfrared/nBrightness <-> Channel Infrared/VICH_PULSE Outputs/nBrightness
//     PlcTask Outputs/GVL_Components.fbMachine.fbVsSystem.fbIllumination2.ChannelInfrared/nDuration_1us <-> Channel Infrared/VICH_PULSE Outputs/nDuration_1us
//     PlcTask Outputs/GVL_Components.fbMachine.fbVsSystem.fbIllumination2.ChannelOrange/nBrightness <-> Channel Orange/VICH_PULSE Outputs/nBrightness
//     PlcTask Outputs/GVL_Components.fbMachine.fbVsSystem.fbIllumination2.ChannelOrange/nDuration_1us <-> Channel Orange/VICH_PULSE Outputs/nDuration_1us
//     PlcTask Outputs/GVL_Components.fbMachine.fbVsSystem.fbIllumination2.DeviceOutputs/bEnable <-> VIMN Outputs Device/bEnable
//     PlcTask Outputs/GVL_Components.fbMachine.fbVsSystem.fbIllumination2.DeviceOutputs/bReset <-> VIMN Outputs Device/bReset
//     PlcTask Outputs/GVL_Components.fbMachine.fbVsSystem.fbIllumination2.Pulse_DC_Outputs/nTimestamp <-> Device/VIOM_PULSE_DC Outputs/nTimestamp
//   Plc/Plc Instance <-> XPlanar MC Project/Axes/Mover4220_1
//     PlcTask Inputs/GVL_Components.fbMachine.aMovers[1].fbMover.MCTOPLC/ACT <-> McToPlc/ACT
//     PlcTask Inputs/GVL_Components.fbMachine.aMovers[1].fbMover.MCTOPLC/COORDMODE <-> McToPlc/COORDMODE
//     PlcTask Inputs/GVL_Components.fbMachine.aMovers[1].fbMover.MCTOPLC/SET <-> McToPlc/SET
//     PlcTask Inputs/GVL_Components.fbMachine.aMovers[1].fbMover.MCTOPLC/SETONTRACK <-> McToPlc/SETONTRACK
//     PlcTask Inputs/GVL_Components.fbMachine.aMovers[1].fbMover.MCTOPLC/STD <-> McToPlc/STD
//     PlcTask Outputs/GVL_Components.fbMachine.aMovers[1].fbMover.PLCTOMC/STD <-> PlcToMc/STD
//   Plc/Plc Instance <-> XPlanar MC Project/Axes/Mover4220_2
//     PlcTask Inputs/GVL_Components.fbMachine.aMovers[2].fbMover.MCTOPLC/ACT <-> McToPlc/ACT
//     PlcTask Inputs/GVL_Components.fbMachine.aMovers[2].fbMover.MCTOPLC/COORDMODE <-> McToPlc/COORDMODE
//     PlcTask Inputs/GVL_Components.fbMachine.aMovers[2].fbMover.MCTOPLC/SET <-> McToPlc/SET
//     PlcTask Inputs/GVL_Components.fbMachine.aMovers[2].fbMover.MCTOPLC/SETONTRACK <-> McToPlc/SETONTRACK
//     PlcTask Inputs/GVL_Components.fbMachine.aMovers[2].fbMover.MCTOPLC/STD <-> McToPlc/STD
//     PlcTask Outputs/GVL_Components.fbMachine.aMovers[2].fbMover.PLCTOMC/STD <-> PlcToMc/STD
//   Plc/Plc Instance <-> XPlanar MC Project/Groups/Environment
//     PlcTask Inputs/GVL_Components.fbMachine.fbXpEnvironment.fbEnvironment.MCTOPLC_STD <-> McToPlc/STD
//   Plc/Plc Instance <-> XPlanar MC Project/Groups/Station1
//     PlcTask Inputs/GVL_Components.fbMachine.fbStation1.fbOptionalTrackUsedInLiveView.MCTOPLC_STD <-> McToPlc/STD
//   Plc/Plc Instance <-> XPlanar MC Project/Groups/Station2
//     PlcTask Inputs/GVL_Components.fbMachine.fbStation2.fbOptionalTrackUsedInLiveView.MCTOPLC_STD <-> McToPlc/STD
//   Plc/Plc Instance <-> XPlanar MC Project/Groups/Station3
//     PlcTask Inputs/GVL_Components.fbMachine.fbStation3.fbOptionalTrackUsedInLiveView.MCTOPLC_STD <-> McToPlc/STD
//   Plc/Plc Instance <-> XPlanar MC Project/Groups/Track1
//     PlcTask Inputs/GVL_Components.fbMachine.fbTrackA.fbTrack.MCTOPLC_STD <-> McToPlc/STD
//   Plc/Plc Instance <-> XPlanar MC Project/Groups/XPlanar
//     PlcTask Inputs/GVL_Components.fbMachine.fbXpGroup.fbGroup.MCTOPLC_STD <-> McToPlc/STD
//   TcCOM Objects/XPlanar/Mover4220_1 <-> XPlanar MC Project/Axes/Mover4220_1
//     InputsFromNC3/NC3ToHW <-> McToIo/STD
//   TcCOM Objects/XPlanar/Mover4220_2 <-> XPlanar MC Project/Axes/Mover4220_2
//     InputsFromNC3/NC3ToHW <-> McToIo/STD
//     OutputsToNC3/HWToNC3 <-> IoToMc/STD
//   Task_IO <-> Device 4 (USB)/Box 2 (C9900-L100 License-Key-USB-Stick)
//     Inputs/Var 2528 <-> BoxInfo/BoxState

CONFIGURATION Plc
    RESOURCE PLC ON TwinCAT3
        TASK PlcTask(INTERVAL := T#1ms, PRIORITY := 5);
        TASK VisionTask(INTERVAL := T#10ms, PRIORITY := 11);
        PROGRAM PRG_ProcessCellSimulation WITH PlcTask : PRG_ProcessCellSimulation;
        PROGRAM PRG_Vision WITH VisionTask : PRG_Vision;
    END_RESOURCE
END_CONFIGURATION

// ---- COMPONENTs/E_ObservationState.TcDUT
{attribute 'qualified_only'}
{attribute 'strict'}
TYPE E_ObservationState :
(
	Idle := 0,
	Observing,
	Qualifying,
	Done
);
END_TYPE

// ---- COMPONENTs/Mode/E_PMLMode.TcDUT
{attribute 'qualified_only'}
TYPE E_PMLMode:
(
	(* Mandatory modes *)
	UNDEFINED := 0,
	PRODUCTION := 1,
	
	(* Optional modes *)
	// MAINTANANCE := 2,
	MANUAL := 3
	
	(* Custom modes *)
	// ?? := 4..32
	// use PML_UnitModeConfig
	
) DINT := UNDEFINED;
END_TYPE

// ---- COMPONENTs/Mode/E_PMLStopReason.TcDUT
{attribute 'qualified_only'}
TYPE E_PMLStopReason :
(
	None := 0,
	Abort_EStop := 1,
	Abort_User := 2,
	Held_Material := 3,
	Held_Ingredients := 4,
	Stop_Actuators := 5,
	Stop_Sensors := 6,
	Suspend_Starved := 7,
	Suspend_Blocked := 8
) DINT := None;
END_TYPE

// ---- COMPONENTs/OEE/ST_Analytics.TcDUT
TYPE ST_Analytics :
STRUCT
	nUnitsProduced : ULINT;
	nDefectiveUnits : ULINT;
	nState : UINT;
	tMlCalculation : TIME;
	bDefectivePart : BOOL;
END_STRUCT
END_TYPE

// ---- COMPONENTs/PackML/ST_PMLc_Custom.TcDUT
TYPE ST_PMLc_Custom EXTENDS ST_PMLcMin :
STRUCT
	Parameter : ARRAY[1..2] OF ST_Descriptor;
END_STRUCT
END_TYPE

// ---- COMPONENTs/PackML/ST_PMLs_Custom.TcDUT
TYPE ST_PMLs_Custom EXTENDS ST_PMLsMin :
STRUCT
	Parameter : ARRAY [1..1] OF ST_Descriptor;
END_STRUCT
END_TYPE

// ---- COMPONENTs/PackML/ST_PML_Custom.TcDUT
TYPE ST_PML_Custom :
STRUCT
	Command 	: ST_PMLc_Custom;
	Status 		: ST_PMLs_Custom;
	Admin 		: ST_PMLaMin;
END_STRUCT
END_TYPE

// ---- COMPONENTs/Vision/E_VisionState.TcDUT
{attribute 'qualified_only'}
{attribute 'strict'}
TYPE E_VisionState :
(
	Idle := 0,
	SelectMode,
	Configure,
	Acquisition,
	Error
);
END_TYPE

// ---- COMPONENTs/Debug.TcGVL
{attribute 'qualified_only'}
VAR_GLOBAL
	tDebug : T_DCTIME64;
	tDebug2 : T_DCTIME64;
	tNow : T_DCTIME64;
END_VAR

// ---- COMPONENTs/GVL_Components.TcGVL
VAR_GLOBAL
	{attribute 'TcContextId':='0'}
	fbMachine : FB_Machine; // Process cell
END_VAR

// ---- COMPONENTs/Vision/I_VsSystem_Check.TcIO
INTERFACE I_VsSystem_Check

METHOD GetQualityRating : I_CH_Feedback
VAR_INPUT
	nDcTrigger : T_DCTIME64;
	nNbrHoles_Expected : LREAL;
	fHoleDiameter : LREAL;
END_VAR
VAR_OUTPUT
	bQualityGood : BOOL;
	nNbrHoles_Found : LREAL;
END_VAR
END_METHOD

END_INTERFACE

// ---- COMPONENTs/Vision/I_VsSystem_Plc.TcIO
INTERFACE I_VsSystem_Plc

METHOD Initialize : HRESULT
VAR_INPUT
END_VAR
END_METHOD

PROPERTY Initialized : BOOL
GET
END_GET
END_PROPERTY

METHOD Update : HRESULT
VAR_INPUT
END_VAR
END_METHOD

METHOD UpdateSlow : HRESULT
VAR_INPUT
END_VAR
END_METHOD

END_INTERFACE

// ---- THREADs/PRG_ProcessCellSimulation.TcPOU
PROGRAM PRG_ProcessCellSimulation

fbMachine.Update();

END_PROGRAM

// ---- THREADs/PRG_Vision.TcPOU
PROGRAM PRG_Vision

fbMachine.UpdateSlow();

END_PROGRAM

// ---- COMPONENTs/FB_Machine.TcPOU
{attribute 'no_explicit_call' := 'do not call this POU directly'} 
FUNCTION_BLOCK FB_Machine EXTENDS FB_Unit
VAR CONSTANT
	N_NBR_MOVERS : UINT := 2;	

	(*	Unique station identification 
		Station ID *)
	S_STATION_NAME_1 : STRING(20) := 'Load';
	S_STATION_NAME_2 : STRING(20) := 'Camera';
	S_STATION_NAME_3 : STRING(20) := 'Unload';
END_VAR
VAR
	(* 	XPlanar System - 1 per associated XPlanar 
		The system is the container and organizer for all subsequent XPlanar objects. 
		All objects are registered with this system	*)
	fbXpSystem 		: FB_XP_System();
	iXpSystem_Plc 	: I_XP_System_PLC := fbXpSystem; 
	
	(* 	XPlanar Collision Avoidance Groupe - 1 per associated XPlanar 
		The Planar group is a software object that prevents collisions between Planar movers as well as collisions of Planar movers with the boundary of 
		the stator area on the two-dimensional XPlanar stator area. To do this, the 2D areas of all objects in the group are blocked. When a motion command 
		is transferred to a mover, the required area is requested from the Planar group and the motion command is rejected if this area would collide 
		with already reserved areas. If the motion command can be executed, the area is added to the set of reserved area and blocked accordingly.	*)
	fbXpGroup : FB_XP_Group(ipSystem := fbXpSystem);
		
	(* 	XPlanar Environment - 1 per associated XPlanar 
		The Planar environment is a software object that represents the two-dimensional XPlanar stator surface. Together with Planar movers in a group, 
		it prevents collisions of the movers with the edge of the surface. *)
	fbXpEnvironment : FB_XP_Environment(ipSystem := fbXpSystem);	
	
	(* 	XPlanar mover - n per associated XPlanar. Can be instantiated as an array and/or individually
		The Planar mover is a software object that represents an XPlanar mover. It summarizes the state of the real mover (position, velocity, etc.) 
		for the user. In addition, the user has the possibility to influence or control the state of the real mover via the Planar mover. *)								
	aMovers : ARRAY[1..N_NBR_MOVERS] OF FB_XP_Mover[
		(ipSystem := fbXpSystem),
		(ipSystem := fbXpSystem)];
	
	(* 	XPlanar track - n per associated XPlanar. Can be instantiated as an array and/or individually
		The Planar track is a software object that represents a (virtual) one-dimensional path on the two-dimensional XPlanar stator surface. 
		Several Planar movers can be lined up and moved on this path. Collisions are prevented by keeping a preset distance between the movers. *)		
	fbTrackA : FB_XP_Track(ipSystem	:= fbXpSystem);	
		
	(* 	XPlanar station - n per associated XPlanar. Can be instantiated as an array and/or individually
		The stations are the main component of the application. As soon as the system has been started up and all movers are on the track, the movers are only sent from one station to the next.
		Parameters:
			xPos, yPos 			= Absolute position of the station on the xPlanar.
			ipAccocietedTrack 	= The track on which the station is located. If the XY position is not on this track, the next possible track position is assumed on this track.
			sStationID 			= Unique name that may only exist once.
			sStationGroupID 	= A name for a group to which this station belongs. Important for redundant stations
			StationAheadx 		= Which station can be approached directly from this station in the positive direction? After a switch there are several possibilities. *)		
	fbStation1	: FB_XP_Station(
					ipSystem := fbXpSystem,
					ipAccocietedTrack := fbTrackA,
					sUniqueName := S_STATION_NAME_1,
					sTargetGroup := '',
					nMoverQueueSize	:= 1,
					xPos := 120,
					yPos := 60);
							
	fbStation2 	: FB_XP_Station(
					ipSystem := fbXpSystem,
					ipAccocietedTrack := fbTrackA,
					sUniqueName := S_STATION_NAME_2,
					sTargetGroup := '',
					nMoverQueueSize := 1,
					xPos := 60,
					yPos := 240);			
	
	fbStation3 	: FB_XP_Station(
					ipSystem := fbXpSystem,
					ipAccocietedTrack := fbTrackA,
					sUniqueName := S_STATION_NAME_3,
					sTargetGroup := '',
					nMoverQueueSize	:= 1,
					xPos := 120,
					yPos := 420);

	(* 	Vision system
		Camera, illumination, trigger, image processing *)								
	fbVsSystem 		: FB_VsSystem;
	iVsSystem_Plc 	: I_VsSystem_Plc := fbVsSystem;
	
	(* 	Machine speed controller
		Controls movement speed based on commanded ppm *)		
	stTaskInfoData : PlcTaskSystemInfo;
	fbSpeedController : FB_Ctrl_PI;
	stSpeedController_Params : ST_Ctrl_PI_Params := (
								bARWOnIPartOnly:= FALSE,
								fOutMinLimit := 100,
								fOutMaxLimit := 1000,
								fKp := 15,
								tTn := T#40S);
	fbRollingAveragePpm : FB_RollingAverage_Ppm;

	(*	Process control variables *)				
	bGetNextProduct : BOOL; // Get next product in manual mode

	(*  The mover leaving station 1 is under observation
		to detect its arrival in the fly-by station 2 (Camera) *)
	bMoverIsObserved : BOOL;
	iMoverObserved : I_XP_Mover_PLC;
	
	eObservationState : E_ObservationState;
	iMoverObserved_Feedback : I_CH_Feedback;
END_VAR

VAR PERSISTENT
	(* 	Analytics
		Overall Equipment Efficiency
		ML Calculation time *)		
	{attribute 'TcAnalytics'}
	{attribute 'OPC.UA.DA' := '1'}	
	stAnalytics : ST_Analytics;		
END_VAR

METHOD PROTECTED Execute_Observation : I_CH_Feedback
VAR CONSTANT
	NBR_CYCLES_AHEAD : UINT := 20; // At least 3.5ms to fit camera requirement
END_VAR
VAR_IN_OUT
	bMoverIsObserved : BOOL;
	iMoverObserved : I_XP_Mover_PLC;
END_VAR
VAR
	(* Calculation of the position window under the camera *)
	fPosition_Mover : LREAL;
	fVelocity_Mover : LREAL;	
	fPosition_Delta : LREAL;
	fPosition_Window : LREAL;
	
	(* Calculation of the time in position *)
	tNow_DC : T_DCTIME64;
	tDelta : ULINT;
	tInPosition_DC : T_DCTIME64;	
END_VAR
VAR_INST
	(* Result Timeout *)
	fbObservationTimeout : TON := (PT:=T#400MS);	
	
	(* Quality feedback *)
	bQualityGood : BOOL;
END_VAR
(* Avoid deadlock if result not present for unloading *)
fbObservationTimeout();
IF fbObservationTimeout.Q THEN
	fbObservationTimeout.IN := FALSE;
	stAnalytics.tMlCalculation := fbObservationTimeout.ET;
	iMoverObserved_Feedback := 0;
	bMoverIsObserved := FALSE;
	iMoverObserved := 0;
	fbRollingAveragePpm.Increment();
	stPackTags.Admin.ProdProcessedCount[1].Count := stPackTags.Admin.ProdProcessedCount[1].Count + 1;
	stPackTags.Admin.ProdDefectiveCount[1].Count := stPackTags.Admin.ProdDefectiveCount[1].Count + 1;
	eObservationState := E_ObservationState.Idle;
END_IF

CASE eObservationState OF
	E_ObservationState.Idle:
		(* Trigger the sequencer *)
		IF bMoverIsObserved AND iMoverObserved <> 0 THEN
			eObservationState := E_ObservationState.Observing;
		END_IF
		
	E_ObservationState.Observing:
		fPosition_Mover := iMoverObserved.PlanarMover.MCTOPLC.SETONTRACK.SetPos; // Store position data 
		fVelocity_Mover := iMoverObserved.PlanarMover.MCTOPLC.SETONTRACK.SetVelo; // Store velocity data		
		fPosition_Delta := iXpSystem_Plc.Station(S_STATION_NAME_2).PositionOnTrack - fPosition_Mover; // Calculate the y position delta
		fPosition_Window := (fVelocity_Mover(*_mm/s*) / 1_000(*_mm/ms*) * (stTaskInfoData.CycleTime / 10_000)(*_mm/cycle*)) * NBR_CYCLES_AHEAD (*_mm*);
		
		(* Leave if mover is not moving *)
		IF (fVelocity_Mover = 0) THEN RETURN; END_IF 
		
		(* Leave if mover is not in window *)
		IF 	fPosition_Window < 0 // Mover direction wrong
		OR 	fPosition_Delta < 0 // Mover already passed camera station
		OR 	ABS(fPosition_Delta) > ABS(fPosition_Window) THEN // Mover not within the window yet
			RETURN;
		END_IF 
		
		(* Predict the time in station with constant velocity *)
		tNow_DC := F_GetCurDcTaskTime64()(*_1ns*);		
		tDelta := TO_ULINT(fPosition_Delta(*_mm*) * 1_000_000_000 / fVelocity_Mover(*_mm/s*));	
		tInPosition_DC := tNow_DC(*_1ns*) + tDelta;
		
		(* Start the visual quality rating *)
		iMoverObserved_Feedback := fbVsSystem.GetQualityRating(
										nDcTrigger:= tInPosition_DC, 
										nNbrHoles_Expected:= stPackTags.Command.Parameter[1].Value, 
										fHoleDiameter:= stPackTags.Command.Parameter[2].Value, 
										bQualityGood=> bQualityGood, 
										nNbrHoles_Found=> stPackTags.Status.Parameter[1].Value);
			
		fbObservationTimeout.IN := TRUE;	
		eObservationState := E_ObservationState.Qualifying;
			
	E_ObservationState.Qualifying:
		(* 	If the quality rating is done
			Store product rating *)
		IF iMoverObserved_Feedback <> 0 AND_THEN iMoverObserved_Feedback.Done THEN
			iMoverObserved_Feedback := 0;
			bMoverIsObserved := FALSE;
			iMoverObserved := 0;
			fbRollingAveragePpm.Increment();	
			
			IF bQualityGood THEN
				stPackTags.Admin.ProdProcessedCount[1].Count := stPackTags.Admin.ProdProcessedCount[1].Count + 1;
			ELSE
				stPackTags.Admin.ProdProcessedCount[1].Count := stPackTags.Admin.ProdProcessedCount[1].Count + 1;
				stPackTags.Admin.ProdDefectiveCount[1].Count := stPackTags.Admin.ProdDefectiveCount[1].Count + 1;
				stAnalytics.bDefectivePart := TRUE;
			END_IF

			fbObservationTimeout.IN := FALSE;
			stAnalytics.tMlCalculation := fbObservationTimeout.ET;
			eObservationState := E_ObservationState.Done;
		END_IF
	
	E_ObservationState.Done:
		eObservationState := E_ObservationState.Idle;
		stAnalytics.bDefectivePart := FALSE;
END_CASE
END_METHOD

{attribute 'object_name' := 'M_Aborting'}
METHOD M_Aborting
VAR_INST
	iFeedback : I_CH_Feedback;
END_VAR
(* Disable XPlanar system if still enabled *)
IF iFeedback = 0 THEN
	iFeedback := iXpSystem_Plc.Disable();
END_IF

(* 	If XPlanar is disabled
	Report stop reason and pause ppm counter *)
IF iFeedback.Done THEN
	stPackTags.Admin.StopReason[1].ID := E_PMLStopReason.None; // Stop reason not specified	
	fbRollingAveragePpm.Enable := FALSE;
	iFeedback := 0;
	M_StateComplete();
END_IF
END_METHOD

{attribute 'object_name' := 'M_Execute'}
METHOD M_Execute
(* 	Apply production speed setpoint in ppm *)
fbSpeedController.fActualValue := fbRollingAveragePpm.Count;
stPackTags.Status.CurMachineSpeed := fbRollingAveragePpm.Count;
fbSpeedController.fSetpointValue := stPackTags.Command.MachSpeed;

(* 	Production speed controller is only active in production mode *)
IF 	stPackTags.Status.UnitModeCurrent = TO_DINT(E_PMLMode.PRODUCTION) 
AND fbRollingAveragePpm.Initialized THEN
		fbSpeedController.eMode := E_CTRL_MODE.eCTRL_MODE_ACTIVE;
ELSE
		(* 	In other modes the setpoint is open loop with default proportional gain (kp)*)
		aMovers[1].SetDynConstraint_Path(stPackTags.Command.MachSpeed * stSpeedController_Params.fKp, 10_000, 10_000, 100_000);
		aMovers[2].SetDynConstraint_Path(stPackTags.Command.MachSpeed * stSpeedController_Params.fKp, 10_000, 10_000, 100_000);
END_IF

(* 	Production speed controller saturation (limit)*)
IF fbSpeedController.fOut < 100 THEN
	aMovers[1].SetDynConstraint_Path(100, 10_000, 10_000, 100_000);
	aMovers[2].SetDynConstraint_Path(100, 10_000, 10_000, 100_000);	

ELSIF fbSpeedController.fOut > 900 THEN
	aMovers[1].SetDynConstraint_Path(900, 10_000, 10_000, 100_000);
	aMovers[2].SetDynConstraint_Path(900, 10_000, 10_000, 100_000);
ELSE
	aMovers[1].SetDynConstraint_Path(fbSpeedController.fOut, 10_000, 10_000, 100_000);
	aMovers[2].SetDynConstraint_Path(fbSpeedController.fOut, 10_000, 10_000, 100_000);
END_IF

IF fbSpeedController.fActualValue > fbSpeedController.fSetpointValue * 1.2 THEN
	fbSpeedController.eMode := E_CTRL_MODE.eCTRL_MODE_RESET;
END_IF

(* Process movers in station 1 *)
IF (iXpSystem_Plc.Station(S_STATION_NAME_1).MoversInPlace) THEN
	IF (stPackTags.Status.UnitModeCurrent = TO_DINT(E_PMLMode.PRODUCTION)) THEN	
		iMoverObserved := iXpSystem_Plc.Station(S_STATION_NAME_1).MoversInQueue[0]; // Start to observe the mover
		bMoverIsObserved := TRUE;
		iXpSystem_Plc.Station(S_STATION_NAME_1).SendMoversToStation(S_STATION_NAME_3); // Send mover directly to the unload station
	ELSIF (stPackTags.Status.UnitModeCurrent = TO_DINT(E_PMLMode.MANUAL) ) THEN
		iXpSystem_Plc.Station(S_STATION_NAME_1).SendMoversToStation(S_STATION_NAME_2); // Send mover into the camera station
	ELSE
		iXpSystem_Plc.Station(S_STATION_NAME_1).SendMoversToStation(S_STATION_NAME_3); // Send mover to avoid deadlock
	END_IF
END_IF

(* Process mover under observation *)
THIS^.Execute_Observation(bMoverIsObserved, iMoverObserved);

(* 	Process movers in station 2 
	only required in manual mode *)
IF (iXpSystem_Plc.Station(S_STATION_NAME_2).MoversInPlace AND bGetNextProduct) THEN
	bGetNextProduct := FALSE;
	iXpSystem_Plc.Station(S_STATION_NAME_2).SendMoversToStation(S_STATION_NAME_3);
END_IF

(* 	Process movers in station 3 
	Touch and go to indicate unload station *)
IF (iXpSystem_Plc.Station(S_STATION_NAME_3).MoversInPlace) THEN
	iXpSystem_Plc.Station(S_STATION_NAME_3).SendMoversToStation(S_STATION_NAME_1);
END_IF
END_METHOD

{attribute 'object_name' := 'M_Resetting'}
METHOD M_Resetting
(* Reset stop reason and equipment interlock *)
stPackTags.Admin.StopReason[1].ID:= E_PMLStopReason.None;
stPackTags.Status.EquipmentInterlock.Blocked := FALSE;
stPackTags.Status.EquipmentInterlock.Starved := FALSE;

(* Reset machine speed control *)
stPackTags.Command.MachSpeed := 20;
fbSpeedController.eMode := E_CTRL_MODE.eCTRL_MODE_RESET;
fbSpeedController.fSetpointValue := stPackTags.Command.MachSpeed;

(* Reset the demo pack tags *)
stPackTags.Command.Parameter[1].ID := 758;
stPackTags.Command.Parameter[1].Name := 'expected_number_of_holes';
stPackTags.Command.Parameter[1].Unit := 'none';
stPackTags.Command.Parameter[1].Value := 8;

stPackTags.Command.Parameter[2].ID := 759;
stPackTags.Command.Parameter[2].Name := 'diameter_of_drillhole';
stPackTags.Command.Parameter[2].Unit := 'mm';
stPackTags.Command.Parameter[2].Value := 5;

stPackTags.Status.Parameter[1].ID := 941;
stPackTags.Status.Parameter[1].Name := 'number_of_correct_holes';
stPackTags.Status.Parameter[1].Unit := 'none';
stPackTags.Status.Parameter[1].Value := 0;

(* Release observed mover*)
bMoverIsObserved := FALSE;
iMoverObserved := 0;
eObservationState := E_ObservationState.Idle;
iMoverObserved_Feedback := 0;

M_StateComplete();
END_METHOD

{attribute 'object_name' := 'M_Starting'}
METHOD M_Starting
VAR_INST
	iFeedback : I_CH_Feedback;
END_VAR
(* Enable XPlanar system if still enabled *)
IF iFeedback = 0 THEN
	iFeedback := iXpSystem_Plc.Enable();
END_IF

(* 	If XPlanar is enabled
	Start ppm counter *)
IF iFeedback <> 0 AND_THEN iFeedback.Done THEN
	fbRollingAveragePpm.Enable := TRUE;
	iFeedback := 0;
	M_StateComplete();
END_IF

(* 	If XPlanar enable failed
	Request machine to abort *)
IF iFeedback <> 0 AND_THEN iFeedback.Error THEN
	fbStateManager(eMode	:= nMode, eCommand := E_PMLState.ePMLState_Aborting, eState	=> eState);
	iFeedback := 0;
END_IF
END_METHOD

{attribute 'object_name' := 'M_Stopping'}
METHOD M_Stopping
VAR_INST
	iFeedback : I_CH_Feedback;
END_VAR
(* Disable XPlanar system if still enabled *)
IF iFeedback = 0 THEN
	iFeedback := iXpSystem_Plc.Disable();
END_IF

(* 	If XPlanar is disabled
	Report stop reason and pause ppm counter *)
IF iFeedback.Done THEN
	stPackTags.Admin.StopReason[1].ID := E_PMLStopReason.Stop_Actuators;
	fbRollingAveragePpm.Enable := FALSE;
	iFeedback := 0;
	M_StateComplete();
END_IF
END_METHOD

METHOD Update
(* Update the unit implementation *)
SUPER^();

(* Update the xplanar *)
IF NOT iXpSystem_Plc.Initialized THEN
	iXpSystem_Plc.Initialize();
ELSE
	iXpSystem_Plc.Update();
END_IF

(* Update the vision system *)
IF NOT iVsSystem_Plc.Initialized THEN
	iVsSystem_Plc.Initialize();
ELSE
	iVsSystem_Plc.Update();
END_IF

(* Update the machine speed controller *)
stTaskInfoData := _TaskInfo[GETCURTASKINDEXEX()];
stSpeedController_Params.tTaskCycleTime := TO_TIME(stTaskInfoData.CycleTime(*_100ns*)/10_000(*_ms*));
stSpeedController_Params.tCtrlCycleTime := T#1S;
fbSpeedController(stParams:=stSpeedController_Params);
fbRollingAveragePpm();

(* Update the analytics statistic *)
stAnalytics.nDefectiveUnits := TO_ULINT(stPackTags.Admin.ProdDefectiveCount[1].Count);
stAnalytics.nUnitsProduced := TO_ULINT(stPackTags.Admin.ProdProcessedCount[1].Count);
stAnalytics.nState := TO_UINT(stPackTags.Status.StateCurrent);
END_METHOD

METHOD UpdateSlow
VAR_INPUT
END_VAR
iVsSystem_Plc.UpdateSlow();
END_METHOD

END_FUNCTION_BLOCK

// ---- COMPONENTs/Unit/FB_Unit.TcPOU
FUNCTION_BLOCK FB_Unit IMPLEMENTS ITF_UnitState
VAR_INPUT (*  	Remark: Since the structure is not implemented as nested FB instances
				the status tags cannot be protected against external manipulation (read-only)
				thus they shall be overwritten each cycle to keep consistancy 			
		
				Could also be mitigated if proper OPC UA pragmas were applied
				within the structure - would require redefinition of top-level
				struct below 
				*)
	{attribute 'TcAnalytics'}
	{attribute 'OPC.UA.DA' := '1'}	
	stPackTags	: ST_PML_Custom;		// Custom pack tags from project
END_VAR

VAR (* 	Protected internal status
		not accessibly, invisible 
		*)
	{attribute 'hide'}
	nMode	: DINT := E_PMLMode.UNDEFINED; // Actual mode of the Unit
	
	{attribute 'hide'}
	bModeValid : BOOL := FALSE; // Indicate if a valid mode is set
	
	{attribute 'hide'}
	eState	: E_PMLState := ePMLState_Aborted; // Actual state of the Unit
	
	{attribute 'hide'}
	fSpeed_Set : REAL; // Set-value of the machine speed
	
	{attribute 'hide'}
	fSpeed_Act : REAL; // Act-value of the machine speed
END_VAR

VAR (*	Mode handler variables *)
	
	{attribute 'hide'}
	fbModeManager : PML_UnitModeManager; // Encapsulated mode change logic
	
	{attribute 'hide'}
	eModeHandler_State : (Wait_For_Change_Request, Switch_Mode, Report_Error); // Method state machine
END_VAR

VAR (*	State handler variables *)
	
	{attribute 'hide'}
	fbStateManager : PML_StateMachine;
END_VAR

(* Refesh the status tags *)
SetTags();

(* Handle mode requests and perform changes *)
ModeHandler();

(* Handle the state if in an valid mode *)
IF bModeValid THEN
	StateHandler();
END_IF

(* Handle the speed request *)
SpeedHandler();

{attribute 'object_name' := 'M_Aborted'}
METHOD M_Aborted
END_METHOD

{attribute 'object_name' := 'M_Aborting'}
METHOD M_Aborting
stPackTags.Admin.StopReason[1].ID := E_PMLStopReason.Abort_User;
M_StateComplete();
END_METHOD

{attribute 'object_name' := 'M_Clearing'}
METHOD M_Clearing
M_StateComplete();
END_METHOD

{attribute 'object_name' := 'M_Complete'}
METHOD M_Complete
END_METHOD

{attribute 'object_name' := 'M_Completing'}
METHOD M_Completing
M_StateComplete();
END_METHOD

{attribute 'object_name' := 'M_Execute'}
METHOD M_Execute
END_METHOD

{attribute 'object_name' := 'M_Held'}
METHOD M_Held
END_METHOD

{attribute 'object_name' := 'M_Holding'}
METHOD M_Holding
stPackTags.Admin.StopReason[1].ID:= E_PMLStopReason.Held_Ingredients;
M_StateComplete();
END_METHOD

{attribute 'object_name' := 'M_Idle'}
METHOD M_Idle
END_METHOD

{attribute 'object_name' := 'M_Resetting'}
METHOD M_Resetting
stPackTags.Admin.StopReason[1].ID:= E_PMLStopReason.None;
stPackTags.Status.EquipmentInterlock.Blocked := FALSE;
stPackTags.Status.EquipmentInterlock.Starved := FALSE;
M_StateComplete();
END_METHOD

{attribute 'object_name' := 'M_Starting'}
METHOD M_Starting
M_StateComplete();
END_METHOD

{attribute 'object_name' := 'M_StateComplete'}
METHOD M_StateComplete
//the actual state is completed
fbStateManager.M_StateComplete();
END_METHOD

{attribute 'object_name' := 'M_Stopped'}
METHOD M_Stopped
END_METHOD

{attribute 'object_name' := 'M_Stopping'}
METHOD M_Stopping
stPackTags.Admin.StopReason[1].ID := E_PMLStopReason.Stop_Actuators;
M_StateComplete();
END_METHOD

{attribute 'object_name' := 'M_Suspended'}
METHOD M_Suspended
END_METHOD

{attribute 'object_name' := 'M_Suspending'}
METHOD M_Suspending
stPackTags.Admin.StopReason[1].ID := E_PMLStopReason.Suspend_Blocked;
stPackTags.Status.EquipmentInterlock.Blocked := TRUE;
M_StateComplete();
END_METHOD

{attribute 'object_name' := 'M_Undefined'}
METHOD M_Undefined
END_METHOD

{attribute 'object_name' := 'M_Unholding'}
METHOD M_Unholding
stPackTags.Admin.StopReason[1].ID := E_PMLStopReason.None;
M_StateComplete();
END_METHOD

{attribute 'object_name' := 'M_Unsuspending'}
METHOD M_Unsuspending
stPackTags.Admin.StopReason[1].ID := E_PMLStopReason.None;
stPackTags.Status.EquipmentInterlock.Blocked := FALSE;
M_StateComplete();
END_METHOD

{attribute 'object_name' := 'ModeHandler'}
METHOD PROTECTED ModeHandler
CASE eModeHandler_State OF
	Wait_For_Change_Request:
		IF stPackTags.Command.UnitModeChangeRequest = TRUE
		AND stPackTags.Command.UnitMode <> E_PMLMode.UNDEFINED
		AND stPackTags.Command.UnitMode <> nMode THEN
			bModeValid := FALSE;
			fbModeManager.eModeCommand := stPackTags.Command.UnitMode;
			eModeHandler_State := Switch_Mode;
		END_IF
		
	Switch_Mode:
		fbModeManager.bExecute := TRUE;
		
		IF fbModeManager.bDone THEN
			bModeValid := TRUE;
			fbModeManager.bExecute := FALSE;
			eModeHandler_State := Wait_For_Change_Request;
			
		ELSIF fbModeManager.bError THEN
			fbModeManager.bExecute := FALSE;
			eModeHandler_State := Report_Error;
		END_IF
		
	Report_Error:
		;
		// Set the machine on fire to highlight urgency
END_CASE

(* 	Execute the mode manager
	and update the status*)
fbModeManager( eState := eState, eModeStatus => nMode);
stPackTags.Status.UnitModeCurrent := nMode;
END_METHOD

{attribute 'object_name' := 'SetTags'}
METHOD PROTECTED SetTags
VAR_INPUT
END_VAR
stPackTags.Status.MachineSpeed := 100;
stPackTags.Status.CurMachineSpeed := 0;
stPackTags.Status.UnitModeCurrent := 0;
END_METHOD

{attribute 'object_name' := 'SpeedHandler'}
METHOD PROTECTED SpeedHandler
VAR_INPUT
END_VAR
(* 	Leave if machine speed mateches the request *)
IF fSpeed_Set = stPackTags.Command.MachSpeed THEN
	RETURN;
END_IF

(*	Apply machine speed within the machines limitations *)
IF stPackTags.Command.MachSpeed <= stPackTags.Status.MachineSpeed THEN
	fSpeed_Set := stPackTags.Command.MachSpeed;
ELSE
	fSpeed_Set := stPackTags.Status.MachineSpeed;
END_IF
END_METHOD

{attribute 'object_name' := 'StateHandler'}
METHOD PROTECTED StateHandler
IF stPackTags.Command.CmdChangeRequest = TRUE THEN
	(* 	Execute the state manager
		and update the status *)
	fbStateManager(eMode	:= nMode, eCommand := stPackTags.Command.CntrlCmd, eState	=> eState);
	stPackTags.Status.StateCurrent := eState;
END_IF

IF stPackTags.Status.UnitModeCurrent <> E_PMLMode.UNDEFINED AND stPackTags.Status.StateCurrent = E_PMLState.ePMLState_Undefined THEN
	stPackTags.Command.CmdChangeRequest := TRUE;
	fbStateManager(eMode	:= nMode, eCommand := E_PMLCommand.ePMLCommand_Abort, eState => eState);
END_IF

IF fbStateManager.bError THEN
	// Set the machine on fire to highlight urgency
END_IF

(*	Process the state method *)
CASE eState OF
	ePMLState_Undefined: M_Undefined();
	ePMLState_Clearing: M_Clearing();
	ePMLState_Stopped: M_Stopped();
	ePMLState_Starting: M_Starting();
	ePMLState_Idle: M_Idle();
	ePMLState_Suspended: M_Suspended();
	ePMLState_Execute: M_Execute();
	ePMLState_Stopping: M_Stopping();
	ePMLState_Aborting: M_Aborting();
	ePMLState_Aborted: M_Aborted();
	ePMLState_Holding: M_Holding();
	ePMLState_Held: M_Held();
	ePMLState_Unholding: M_Unholding();
	ePMLState_Suspending: M_Suspending();
	ePMLState_Unsuspending: M_Unsuspending();
	ePMLState_Resetting: M_Resetting();
	ePMLState_Completing: M_Completing();
	ePMLState_Complete: M_Complete();
END_CASE
END_METHOD

END_FUNCTION_BLOCK

// ---- COMPONENTs/Vision/FB_VsSystem.TcPOU
{attribute 'no_explicit_call' := 'do not call this POU directly'} 
FUNCTION_BLOCK FB_VsSystem IMPLEMENTS I_VsSystem_Check, I_VsSystem_Plc
VAR CONSTANT
	(* Machine learning model constants *)
	N_MODEL_NBR_INPUT_CHANNELS: UDINT := 3;
	N_MODEL_INPUT_WIDTH: 		UDINT := 224;
	N_MODEL_INPUT_HEIGHT: 		UDINT := 224;
	N_MODEL_NBR_CLASSES: 		UDINT := 2; // ADJUST NUMBER OF CLASSES WHEN CHANGING MODEL!!!
	N_MAX_PIXEL_VALUE: 			UDINT := 255;
	
	(* Preprocessing constants *)
	N_RESIZE_WIDTH				: UDINT := 256;
	N_RESIZE_HEIGHT				: UDINT := 256;
	N_CENTRAL_CROPPING_WIDTH	: UDINT := 224;
	N_CENTRAL_CROPPING_HEIGHT	: UDINT := 224;
	
	(* Contour filter criteria *) 
	F_MINLENGTHCONTOUR			: LREAL := 5700; 
	F_MINAREACONTOUR			: LREAL := 1050000; 
	
END_VAR

VAR
	fbFeedback 					: FB_CH_Feedback(0);
	
	(* Vision system and its components *)
	fbImageProvider 			: FB_GigE_Beckhoff();
	fbCameraTriggerController	: FB_EtherCAT_Trigger;
	fbIllumination1				: FB_VIx2000();
	fbIllumination2				: FB_VIx2000();
	fbPulseMode 				: FB_VisionMode_Pulse_combined;
	
	fbVisionSystemCHALET 		: FB_VisionSystem(
									ipImageProvider				:= fbImageProvider, 
									ipCameraTriggerController 	:= fbCameraTriggerController, 
									ipIlluminationController1 	:= fbIllumination1, 
									ipIlluminationController2 	:= fbIllumination2);
										
	iVisionSystem 				: I_VisionSystem := fbVisionSystemCHALET;
	
	(* Puls Settings *)
	nOrange 					: UINT(0..511) 	:= 511; 
	nGreen 						: UINT(0..511)	:= 511;
	nBlue 						: UINT(0..511) 	:= 511;	
	nInfrared 					: UINT(0..511)	:= 511; 
	nExposure_1us 				: UDINT := 50; 
	nExposureDelay_100ns		: UDINT := 10;
	nIlluminationOverride   	: USINT := 100;
	nIlluminationDuration_1us 	: UDINT := 70; 
	
	(* State machine *)
	eVisionState 				: E_VisionState;	
	hr 							: HRESULT;

	(* Commands *)
	bTrigger,bTriggerNonStop	: BOOL;
	bPulsMode					: BOOL := TRUE;
	bCustomerMode				: BOOL;
	bApply						: BOOL;	
	bTriggerFixRate				: BOOL;
	nFixRateDelayMs 			: UINT := 10;
	nNextCamTrigger				: T_DCTIME64;
	nNextIllTrigger				: T_DCTIME64;
		
	(* Interface to image processing *)
	SLOW_hrGlobal 				: HRESULT;
	SLOW_nImageCounter 			: UDINT;
	SLOW_ipLiveImgWithInfo 		: ST_ImageWithInfo;
	SLOW_ipDispImageInRGB 		: ITcVnDisplayableImage;
	
	fbCrititcalSection 			: FB_IecCriticalSection;
	
	(* Interface to machine*)
	bQualityGood				: BOOL;
	nNbrHoles_Expected 			: ULINT;
	fHoleDiameter 				: LREAL;
	nNbrHoles_Found 			: ULINT;
END_VAR

METHOD GetQualityRating : I_CH_Feedback
VAR_INPUT
	nDcTrigger : T_DCTIME64;
	nNbrHoles_Expected : LREAL;
	fHoleDiameter : LREAL;
END_VAR
VAR_OUTPUT
	bQualityGood : BOOL;
	nNbrHoles_Found : LREAL;
END_VAR
VAR
	hr : HRESULT;
END_VAR
IF fbCrititcalSection.Enter() THEN
	(* Transfer recipe command parameters *)
	THIS^.nNbrHoles_Expected := TO_ULINT(nNbrHoles_Expected);
	THIS^.fHoleDiameter := fHoleDiameter;	
	(* end of critical section *)
	fbCrititcalSection.Leave();
END_IF

IF iVisionSystem.Operational AND NOT iVisionSystem.Busy THEN
	hr := fbPulseMode.TriggerAtDcTime(nDcTrigger);
	
	IF fbCrititcalSection.Enter() THEN
		(* start of critical section *)
		fbFeedback.Busy := TRUE;
		(* end of critical section *)
		fbCrititcalSection.Leave();
	END_IF
END_IF

IF fbCrititcalSection.Enter() THEN
	(* Transfer recipe status parameters *)
	nNbrHoles_Found := TO_REAL(THIS^.nNbrHoles_Found);
	(* Transfer result *)
	bQualityGood := THIS^.bQualityGood;
	(* start of critical section *)
	GetQualityRating := fbFeedback;
	(* end of critical section *)
	fbCrititcalSection.Leave();
END_IF
END_METHOD

METHOD Initialize : HRESULT
VAR_INPUT
END_VAR
IF fbVisionSystemCHALET.Initialized THEN
	
	Initialize := S_OK;
ELSE
	fbVisionSystemCHALET.Initialize();
	Initialize := S_PENDING;
END_IF
END_METHOD

{attribute 'monitoring' := 'call'}
PROPERTY Initialized : BOOL
GET
Initialized := fbVisionSystemCHALET.Initialized;
END_GET
END_PROPERTY

METHOD Update : HRESULT
CASE eVisionState OF
	E_VisionState.Idle:
		eVisionState := E_VisionState.SelectMode;
	
	E_VisionState.SelectMode:
		hr := iVisionSystem.SetMode(fbPulseMode);
		
		IF hr = S_OK THEN
			eVisionState := E_VisionState.Configure;
		ELSIF FAILED(hr) OR iVisionSystem.Error THEN
			eVisionState := E_VisionState.Error;	
		END_IF
	
	(* Initial configuration during start-up *)
	E_VisionState.Configure:
		hr := fbPulseMode.Configure(nOrange := nOrange,	// 0-511
									nGreen := nGreen,	// 0-511
									nBlue := nBlue,	// 0-511
									nInfrared := nInfrared, // 0-511
									nExposure_1us := nExposure_1us,
									nIlluminationOverride := nIlluminationOverride(*1-100*),
									nIlluminationDuration_1us := nIlluminationDuration_1us);
									
			
		IF hr = S_OK THEN
			eVisionState := E_VisionState.Acquisition;
		ELSIF FAILED(hr) OR iVisionSystem.Error THEN
			eVisionState := E_VisionState.Error;		
		END_IF
		
	(* Re-configuration during acquisition *)
	E_VisionState.Acquisition:
		IF bApply THEN
			bApply := FALSE;
			eVisionState := E_VisionState.Configure;
		END_IF		
		
		IF FAILED(hr) OR iVisionSystem.Error THEN
			eVisionState := E_VisionState.Error;		
		END_IF
		
	E_VisionState.Error:
		hr := iVisionSystem.Reset();
		eVisionState := E_VisionState.Idle;

END_CASE

iVisionSystem.Update();
END_METHOD

METHOD UpdateSlow : HRESULT
VAR_INST
	_ImageAvailable 				: BOOL;
	
	//ML Variables
	hr_predict						: HRESULT;
	// Load Model

	sFolderPath						: STRING(255) := 'C:\Technology_Update_2024\Day2_QualityCheck\ML_models\model_11_72\';
	sFileName						: STRING(255) := 'model_11_72.onnx';
	sFilePath_ML            		: STRING(255) := '';
	
	fbReadDnn						: FB_VN_ReadNeuralNetwork;
	ipDnnModel						: ITcVnNeuralNetwork;
	bDnnModelInitialized			: BOOL := FALSE;
	nReturnCode						: UDINT;
	
	// Model information
	sClassLabels					: ARRAY[0..N_MODEL_NBR_CLASSES] OF STRING := ['nok_kratzer: ', 'ok_surface: ']; // ADJUST CLASS LABELS WHEN CHANGING MODEL!!!
	aStd							: TcVnVector4_LREAL := [0.229, 0.224, 0.225];
	aMean							: TcVnVector4_LREAL := [0.485, 0.456, 0.406];
	ePaddingMode					: ETcVnPaddingMode := TCVN_PM_NONE;
	eInterpolationType				: ETcVnInterpolationType := TCVN_IT_BILINEAR; // Corresponds to cv.INTER_LINEAR
	
	// ML Images
	ipPreprocessedImageIn			: ITcVnImage;
	ipResizedImageInDisp			: ITcVnDisplayableImage;
	ipDispImageMLResult				: ITcVnDisplayableImage;
	stPixelFormat					: TcVnPixelFormat;
	ipTensorImage					: ITcVnImage;
	ipDnnOutputImage				: ITcVnImage;
	
	// Result
	nDnnOutputSize					: ULINT	:= 0;
	aDnnOutputVector 				: ARRAY[1..N_MODEL_NBR_CLASSES] OF REAL; //ARRAY[1..cNumberOfClasses] OF REAL;
	aConfidence						: TcVnVector4_LREAL;
	aClassIndex						: TcVnPoint2_DINT;
	sResult							: STRING(255);
	
	// Classical vision Images
	SLOW_ipImageWork 		: ITcVnImage; //Image to work on
	SLOW_ipDispImageWork 	: ITcVnDisplayableImage; //Displayable image to work on
	SLOW_ipImageWork_old 	: ITcVnImage; //Image to compare with new image

	ipStructuringElement 	: ITcVnImage; //Structuring element
	ipContours 				: ITcVnContainer; //Found contours in image
    ipIterator       		: ITcVnForwardIterator; //Iterator for the contour container
    ipContour        		: ITcVnContainer; //Single contour container
	ipMAXContour			: ITcVnContainer; //MAX contour container
	nNbrOfContours			: ULINT; 
	fContourArea			: LREAL; 
	fMAXContourArea			: LREAL; 

	fMINLimitContourArea	: LREAL := 1_000; //Lower limit of a borehole
	fMAXLimitContourArea	: LREAL := 15_000; //Upper limit of a borehole

	aOffset 				: TcVnPoint := [0, 0];
	aColRed       			: TcVnVector4_LREAL := [255, 0, 0, 255];
	aColGreen        		: TcVnVector4_LREAL := [0, 255, 0, 255];
	aColPink        		: TcVnVector4_LREAL := [255, 100, 255, 255];
	aColBlack        		: TcVnVector4_LREAL := [0, 0, 0, 255];

	fLengthMAXContour		: LREAL; 
	nYLabelPos				: UDINT := 80;
	
	ipFilteredContours 		: ITcVnContainer; //Container containing the contours matching the fMINLimitContourArea and fMAXLimitContourArea criteria
	aImgIntensityAverage   	: TcVnVector4_LREAL;
END_VAR
_ImageAvailable := iVisionSystem.TryGetImage(SLOW_ipLiveImgWithInfo) = S_OK;
// Load Dnn model
IF NOT bDnnModelInitialized THEN
	sFilePath_ML := CONCAT (sFolderPath, sFileName);
	FW_SafeRelease(ADR(ipDnnModel));
	fbReadDnn(sFilePath := sFilePath_ML, ipDestNeuralNetwork := ipDnnModel, bRead := TRUE);

	IF NOT fbReadDnn.bBusy THEN
		fbReadDnn(sFilePath:='', bRead := FALSE);
		IF NOT fbReadDnn.bError THEN
			bDnnModelInitialized := TRUE;
		END_IF
		nReturnCode := fbReadDnn.nErrorId AND 16#FFF;
	END_IF
END_IF
	
IF _ImageAvailable THEN
	SLOW_hrGlobal := S_OK;
	SLOW_nImageCounter := SLOW_nImageCounter + 1;
	fMAXContourArea := 0;
	SLOW_hrGlobal := F_VN_ConvertColorSpace(ipSrcImage:= SLOW_ipLiveImgWithInfo.ipImage, ipDestImage:= SLOW_ipLiveImgWithInfo.ipImage, eTransform:= TCVN_CST_BAYER_RG_TO_GRAY, hrPrev:= SLOW_hrGlobal);
	
	//Create work image to apply vision operations on, leave oringal image unedited 
	SLOW_hrGlobal := F_VN_CopyImage(ipSrcImage:= SLOW_ipLiveImgWithInfo.ipImage, ipDestImage:= SLOW_ipImageWork, hrPrev:= SLOW_hrGlobal);
	
	//////////////////////////////////////////////////////////////
	//////////////////////////////////////////////////////////////
	/////////////////////////ML VISION////////////////////////////
	//////////////////////////////////////////////////////////////
	//////////////////////////////////////////////////////////////
	
	// Check if new image was received
	IF bDnnModelInitialized AND SUCCEEDED(SLOW_hrGlobal) AND SLOW_ipLiveImgWithInfo.ipImage <> 0 THEN
		hr_predict := F_VN_GetPixelFormat(SLOW_ipLiveImgWithInfo.ipImage, stPixelFormat, hr_predict);

		// Check if input image channels matches the model requirements, alternative implement the needed color space transformation yourself.
		IF stPixelFormat.nChannels <> N_MODEL_NBR_INPUT_CHANNELS OR stPixelFormat.ePixelEncoding <> TCVN_PE_NONE THEN
			hr_predict := F_VN_ConvertColorSpace(SLOW_ipLiveImgWithInfo.ipImage, ipPreprocessedImageIn, TCVN_CST_GRAY_TO_RGB, hr_predict);                
		END_IF

		// *** Preprocessing steps ***
		// Adjust the dimensions of the input image to match the model input requirements
		// Resize
		hr_predict := F_VN_ResizeImageExp(ipPreprocessedImageIn, ipPreprocessedImageIn, N_RESIZE_WIDTH, N_RESIZE_HEIGHT, eInterpolationType, ePaddingMode, aColBlack, hr_predict);
			
		// Convert the image to type REAL and scale to the range [0.0, 1.0]
		hr_predict := F_VN_ConvertElementTypeExp(ipPreprocessedImageIn, ipTensorImage, TCVN_ET_REAL, 1.0 / UDINT_TO_REAL(N_MAX_PIXEL_VALUE), 0, hr_predict);

		// Normalization
		hr_predict := F_VN_SubtractVectorFromImage(ipTensorImage, aMean, ipTensorImage,hr_predict);
		hr_predict := F_VN_DivideImageByVector(ipTensorImage, aStd, ipTensorImage, hr_predict);

		// Convert the input image to 4D Tensor
		hr_predict := F_VN_ConvertDataLayout(ipTensorImage, ipTensorImage, TCVN_DL_4D_NCHW, hr_predict);

		// *** Model execution ***
		hr_predict := F_VN_ExecuteNeuralNetwork(ipDnnModel, ipTensorImage, ipDnnOutputImage, hr_predict);
		
		// Export result from NN
		hr_predict := F_VN_ExportImageSize(ipDnnOutputImage, nDnnOutputSize, hr_predict);
		hr_predict := F_VN_ExportImage(ipDnnOutputImage, ADR(aDnnOutputVector), nDnnOutputSize, hr_predict 	);

		// *** Postprocessing steps ***
		// Get best classfication result
		hr_predict := F_VN_MaxPixelValue(ipDnnOutputImage, aConfidence , aClassIndex, hr_predict);

		// Result visualization
		//sResult := CONCAT(CONCAT(CONCAT(sClassLabels[aClassIndex[0]] , LREAL_TO_FMTSTR(aConfidence[0], 2, FALSE)), ' ImgNr. '), TO_STRING(SLOW_nImageCounter));
		//hr_predict := F_VN_PutLabelExp(sResult, SLOW_ipImageWork, 5, 120, 7, 2, TCVN_FT_HERSHEY_PLAIN, aColBlack, aColWhite, TCVN_LT_4_CONNECTED, hr_predict);
		//SLOW_nConfidence := aConfidence[0];
		
		// Display images and release pointer
		hr_predict := F_VN_TransformIntoDisplayableImage(ipPreprocessedImageIn, ipResizedImageInDisp, S_OK);
		hr_predict := F_VN_CopyIntoDisplayableImage(SLOW_ipImageWork, ipDispImageMLResult, S_OK);
		FW_SafeRelease(ADR(ipTensorImage));
		FW_SafeRelease(ADR(ipDnnOutputImage));
	END_IF

	FW_SafeRelease(ADR(SLOW_ipImageWork));

	//Create work image to apply vision operations on, leave oringal image unedited 
	SLOW_hrGlobal := F_VN_CopyImage(ipSrcImage:= SLOW_ipLiveImgWithInfo.ipImage, ipDestImage:= SLOW_ipImageWork, hrPrev:= SLOW_hrGlobal);
	
	//////////////////////////////////////////////////////////////
	//////////////////////////////////////////////////////////////
	//////////////////CLASSICAL VISION////////////////////////////
	//////////////////////////////////////////////////////////////
	//////////////////////////////////////////////////////////////
	
	//smooth image to remove noise
	SLOW_hrGlobal := F_VN_GaussianFilter(
						ipSrcImage:= SLOW_ipImageWork, 
						ipDestImage:= SLOW_ipImageWork, 
						nFilterWidth:= 17, 
						nFilterHeight:= 17, 
						hrPrev:= SLOW_hrGlobal);
	
	//binarize image					
	SLOW_hrGlobal := F_VN_Threshold(
						ipSrcImage:= SLOW_ipImageWork, 
						ipDestImage:= SLOW_ipImageWork, 
						fThreshold:= 25, 
						fMaxValue:= 255, 
						eThresholdType:= TCVN_TT_BINARY, 
						hrPrev:= SLOW_hrGlobal);					
	
	FW_SafeRelease(ADR(ipStructuringElement));	
	
	//apply morphological opening to remove small unwanted holes 			
	SLOW_hrGlobal := F_VN_CreateStructuringElement(
						ipStructuringElement:= ipStructuringElement, 
						eShape:= TCVN_SES_RECTANGLE, 
						nWidth:= 17, 
						nHeight:= 17, 
						hrPrev:= SLOW_hrGlobal);
	
	SLOW_hrGlobal := F_VN_MorphologicalOperator(
						ipSrcImage:= SLOW_ipImageWork, 
						ipDestImage:= SLOW_ipImageWork, 
						eOperator:= TCVN_MO_CLOSING, 
						ipStructuringElement:= ipStructuringElement, 
						hrPrev:= SLOW_hrGlobal);
	
	SLOW_hrGlobal := F_VN_ImageAverage(ipSrcImage:= SLOW_ipImageWork, aAverage:= aImgIntensityAverage, hrPrev:= SLOW_hrGlobal);

	//find contours in the image, using black-white image borders
	SLOW_hrGlobal := F_VN_FindContoursExp(
						ipSrcImage:= SLOW_ipImageWork, 
						ipContours:= ipContours, 
						eRetrievalMode:= TCVN_CRM_LIST, 
						eApproximationMethod:= TCVN_CAM_SIMPLE, 
						aOffset:= aOffset, 
						hrPrev:= SLOW_hrGlobal);
	
	//Count total number of found contours
	SLOW_hrGlobal := F_VN_GetNumberOfElements(ipContainer:= ipContours, nNumberOfElements:= nNbrOfContours, hrPrev:= SLOW_hrGlobal); 
	SLOW_hrGlobal := F_VN_CreateContainer(ipFilteredContours, ContainerType_Vector_Vector_TcVnPoint2_DINT, 0, SLOW_hrGlobal);
	
	SLOW_hrGlobal := F_VN_ConvertColorSpace(ipSrcImage:= SLOW_ipImageWork, ipDestImage:= SLOW_ipImageWork, eTransform:= TCVN_CST_GRAY_TO_RGB, hrPrev:= SLOW_hrGlobal);

	// Initialize the iterator for the ipContours container
	SLOW_hrGlobal := F_VN_GetForwardIterator(ipContours, ipIterator, SLOW_hrGlobal);
	
	// Iterate over the contours in the container
	WHILE SUCCEEDED(SLOW_hrGlobal) AND_THEN ipIterator.CheckIfEnd() <> S_OK DO
		// Get the current contour from the iterator
		hr := F_VN_GetContainer(ipIterator, ipContour, SLOW_hrGlobal);
		
		IF ipContour <> 0 THEN
			SLOW_hrGlobal := F_VN_ContourArea(ipContour:= ipContour, fArea:= fContourArea, hrPrev:= SLOW_hrGlobal);
			
			//Get contour area of biggest contour -> measure if part has correct size 
			IF fContourArea > fMAXContourArea THEN
				fMAXContourArea := fContourArea;
				FW_SafeRelease(ADR(ipMAXContour));
				SLOW_hrGlobal := F_VN_CopyContainer(ipSrcContainer:= ipContour, ipDestContainer:= ipMAXContour, hrPrev:= SLOW_hrGlobal);    
				//F_VN_SetContainer(ipIterator:= ipIterator, ipContainer:= ipMAXContour, hrPrev:= SLOW_hrGlobal);
			END_IF
			
			//Filter the found contours based on contour area -> Limits should only allow for the small boreholes 
			IF (fContourArea > fMINLimitContourArea) AND (fContourArea < fMAXLimitContourArea) THEN 
				SLOW_hrGlobal := F_VN_AppendToContainer_ITcVnContainer(ipElement:= ipContour, ipContainer:= ipFilteredContours, hrPrev:= SLOW_hrGlobal);
			END_IF
		END_IF
		FW_SafeRelease(ADR(ipContour));

		//Increment iterator to the next contour
		SLOW_hrGlobal := F_VN_IncrementIterator(ipIterator, SLOW_hrGlobal);
	END_WHILE
	FW_SafeRelease(ADR(ipIterator));
	
	//Count number of boreholes 
	SLOW_hrGlobal := F_VN_GetNumberOfElements(ipContainer:= ipFilteredContours, nNumberOfElements:= THIS^.nNbrHoles_Found, hrPrev:= SLOW_hrGlobal); 
	
	//Visualize MAX-Contour 
	SLOW_hrGlobal := F_VN_DrawContoursExp(
						ipContours:= ipMAXContour, 
						nContourIndex:= -1, 
						ipDestImage:= SLOW_ipImageWork, 
						aColor:= aColPink, 
						nThickness:= 3, 
						eLineType:= TCVN_LT_4_CONNECTED , 
						ipHierarchy:= 0, 
						nMaxLevel:= 4, 
						aOffset:= aOffset, 
						hrPrev:= SLOW_hrGlobal);
	
	//Visualize boreholes only
	SLOW_hrGlobal := F_VN_DrawContoursExp(
						ipContours:= ipFilteredContours, 
						nContourIndex:= -1, 
						ipDestImage:= SLOW_ipImageWork, 
						aColor:= aColGreen, 
						nThickness:= 3, 
						eLineType:= TCVN_LT_4_CONNECTED , 
						ipHierarchy:= 0, 
						nMaxLevel:= 4, 
						aOffset:= aOffset, 
						hrPrev:= SLOW_hrGlobal);
						
	//Contour analysis					
	SLOW_hrGlobal := F_VN_ContourPerimeter(ipContour:= ipMAXContour, fPerimeter:= fLengthMAXContour, bClosed:= TRUE, hrPrev:= SLOW_hrGlobal);

	//get comprehensive part inspection result ML + clssic CV Results -> OK NOK 
	sResult := CONCAT('# Holes: ', TO_STRING(THIS^.nNbrHoles_Found));
	IF THIS^.nNbrHoles_Found =  THIS^.nNbrHoles_Expected THEN 
		SLOW_hrGlobal := F_VN_PutLabelExp(sResult, SLOW_ipImageWork, 5, nYLabelPos, 7, 2, TCVN_FT_HERSHEY_PLAIN, aColBlack, aColGreen, TCVN_LT_4_CONNECTED, SLOW_hrGlobal);
	ELSE
		SLOW_hrGlobal := F_VN_PutLabelExp(sResult, SLOW_ipImageWork, 5, nYLabelPos, 7, 2, TCVN_FT_HERSHEY_PLAIN, aColBlack, aColRed, TCVN_LT_4_CONNECTED, SLOW_hrGlobal);
	END_IF

	sResult := CONCAT('Length Cnt.: ', LREAL_TO_FMTSTR(fLengthMAXContour, 0, TRUE));
	IF fLengthMAXContour > F_MINLENGTHCONTOUR AND_THEN  fLengthMAXContour < F_MINLENGTHCONTOUR + 400 THEN 
		SLOW_hrGlobal := F_VN_PutLabelExp(sResult, SLOW_ipImageWork, 5, nYLabelPos * 2, 7, 2, TCVN_FT_HERSHEY_PLAIN, aColBlack, aColGreen, TCVN_LT_4_CONNECTED, SLOW_hrGlobal);
	ELSE
		SLOW_hrGlobal := F_VN_PutLabelExp(sResult, SLOW_ipImageWork, 5, nYLabelPos * 2, 7, 2, TCVN_FT_HERSHEY_PLAIN, aColBlack, aColRed, TCVN_LT_4_CONNECTED, SLOW_hrGlobal);
	END_IF
	
	sResult := CONCAT('Area Cnt.: ', LREAL_TO_FMTSTR(fMAXContourArea, 0, TRUE)); 
	IF fMAXContourArea > F_MINAREACONTOUR THEN 
		SLOW_hrGlobal := F_VN_PutLabelExp(sResult, SLOW_ipImageWork, 5, nYLabelPos * 3, 7, 2, TCVN_FT_HERSHEY_PLAIN, aColBlack, aColGreen, TCVN_LT_4_CONNECTED, SLOW_hrGlobal);
	ELSE
		SLOW_hrGlobal := F_VN_PutLabelExp(sResult, SLOW_ipImageWork, 5, nYLabelPos * 3, 7, 2, TCVN_FT_HERSHEY_PLAIN, aColBlack, aColRed, TCVN_LT_4_CONNECTED, SLOW_hrGlobal);
	END_IF
	
	IF sClassLabels[aClassIndex[0]] = 'ok_surface: ' THEN 
		sResult := 'Surface: OK';
		SLOW_hrGlobal := F_VN_PutLabelExp(sResult, SLOW_ipImageWork, 5, nYLabelPos * 4, 7, 2, TCVN_FT_HERSHEY_PLAIN, aColBlack, aColGreen, TCVN_LT_4_CONNECTED, SLOW_hrGlobal);
	ELSE
		sResult := 'Surface: NOK';
		SLOW_hrGlobal := F_VN_PutLabelExp(sResult, SLOW_ipImageWork, 5, nYLabelPos * 4, 7, 2, TCVN_FT_HERSHEY_PLAIN, aColBlack, aColRed, TCVN_LT_4_CONNECTED, SLOW_hrGlobal);
	END_IF

	IF THIS^.nNbrHoles_Found = THIS^.nNbrHoles_Expected AND fLengthMAXContour > F_MINLENGTHCONTOUR AND fMAXContourArea > F_MINAREACONTOUR AND sClassLabels[aClassIndex[0]] = 'ok_surface: ' THEN 
		bQualityGood := TRUE;
		sResult := 'PART OK';
		SLOW_hrGlobal := F_VN_PutLabelExp(sResult, SLOW_ipImageWork, 1900, nYLabelPos, 7, 3, TCVN_FT_HERSHEY_PLAIN, aColBlack, aColGreen, TCVN_LT_4_CONNECTED, SLOW_hrGlobal);
	ELSE
		bQualityGood := FALSE;
		sResult := 'PART NOK';
		SLOW_hrGlobal := F_VN_PutLabelExp(sResult, SLOW_ipImageWork, 1900, nYLabelPos, 7, 3, TCVN_FT_HERSHEY_PLAIN, aColBlack, aColRed, TCVN_LT_4_CONNECTED, SLOW_hrGlobal);
	END_IF
	
	//Free router memory
	FW_SafeRelease(ADR(ipContours));
	FW_SafeRelease(ADR(ipFilteredContours));
	FW_SafeRelease(ADR(SLOW_ipDispImageInRGB));
	FW_SafeRelease(ADR(SLOW_ipDispImageWork));
	FW_SafeRelease(ADR(ipMAXContour));
	FW_SafeRelease(ADR(SLOW_ipImageWork_old));
	
	SLOW_hrGlobal := F_VN_CopyImage(ipSrcImage:= SLOW_ipImageWork, ipDestImage:= SLOW_ipImageWork_old, hrPrev:= SLOW_hrGlobal);
	
	//Transform the two images into displayable images 
	SLOW_hrGlobal := F_VN_TransformIntoDisplayableImage(SLOW_ipLiveImgWithInfo.ipImage, SLOW_ipDispImageInRGB, SLOW_hrGlobal);
	SLOW_hrGlobal := F_VN_TransformIntoDisplayableImage(SLOW_ipImageWork, SLOW_ipDispImageWork, SLOW_hrGlobal);
	
	IF fbCrititcalSection.Enter() THEN
		(* start of critical section *)
		fbFeedback.Done := TRUE;
		(* end of critical section *)
		fbCrititcalSection.Leave();
	END_IF
END_IF
END_METHOD

END_FUNCTION_BLOCK

// ---- COMPONENTs/FB_RollingAverage_Ppm.TcPOU
FUNCTION_BLOCK FB_RollingAverage_Ppm
VAR CONSTANT
	LOW : UINT := 0;
	HIGH : UINT := 59;
END_VAR
VAR
	aCounts : ARRAY[LOW..HIGH] OF UINT;
	fbTimer : TON := (PT:=T#1S);
	nLatestIndex : UINT := LOW;
	bInitialized : BOOL;
	nIdx : UINT;
	bEnable : BOOL;
END_VAR

IF bEnable THEN
	fbTimer(IN := TRUE);
	IF fbTimer.Q THEN
		fbTimer(IN := FALSE);
		aCounts[nLatestIndex] := 0;
		nLatestIndex := (nLatestIndex + 1) MOD (HIGH + 1);
		IF (nLatestIndex = 0) THEN bInitialized := TRUE; END_IF
	END_IF
ELSE
	fbTimer(IN := FALSE);
	nLatestIndex := LOW;
	bInitialized := FALSE;
	FOR nIdx := LOW TO HIGH DO
		aCounts[nIdx] := 0;
	END_FOR
END_IF

{attribute 'monitoring' := 'call'}
PROPERTY Count : UINT
GET
Count := aCounts[nLatestIndex];
END_GET
END_PROPERTY

{attribute 'monitoring' := 'call'}
PROPERTY Enable : BOOL
GET
Enable := bEnable;
END_GET
SET
bEnable := Enable;
END_SET
END_PROPERTY

METHOD Increment
VAR
	nIdx : UINT;
END_VAR
FOR nIdx := LOW TO HIGH DO
	aCounts[nIdx] := aCounts[nIdx] + 1;
END_FOR
END_METHOD

{attribute 'monitoring' := 'call'}
PROPERTY Initialized : BOOL
GET
Initialized := bInitialized;
END_GET
END_PROPERTY

END_FUNCTION_BLOCK
